DATA_BLOCK "METIS_AUX_DB"   // DB100
TITLE = Auxiliary help variables
{ S7_Optimized_Access := 'FALSE' }
AUTHOR : METIS
FAMILY : ACESYS
NAME : MiscDB
VERSION : 8.0
   VAR
      _REAL : Array[1..1000] of Real;   // Temporary REAL variables
      _INT : Array[1..200] of Int;   // Temporary INT variables
      _DINT : Array[1..200] of DInt;   // Temporary DINT variables
      _TIME : Array[1..100] of Time;   // Temporary TIME variables
      _BOOL : Array[1..512] of Bool;   // Temporary BOOLEAN variables
   END_VAR
BEGIN
   _REAL[1] := 8.0;
   _REAL[2] := 0.0;
   _REAL[3] := 16#FFC0_0000;
   _REAL[4] := 0.0;
   _REAL[5] := 0.0;
   _REAL[6] := 360.0;
   _REAL[7] := 1.0;
   _REAL[8] := 0.0;
   _REAL[9] := -32768.0;
   _REAL[10] := 0.0;
   _REAL[11] := 0.0;
   _REAL[12] := 0.0;
   _REAL[13] := 0.0;
   _REAL[14] := 0.0;
   _REAL[15] := 0.0;
   _REAL[16] := 0.0;
   _REAL[17] := 0.0;
   _REAL[18] := 0.0;
   _REAL[19] := 0.0;
   _REAL[20] := 0.0;
   _REAL[21] := 0.0;
   _REAL[22] := 0.0;
   _REAL[23] := 0.0;
   _REAL[24] := 0.0;
   _REAL[25] := 0.0;
   _REAL[26] := 0.0;
   _REAL[27] := 0.0;
   _REAL[28] := 0.0;
   _REAL[29] := 0.0;
   _REAL[30] := 0.0;
   _REAL[31] := 0.0;
   _REAL[32] := 0.0;
   _REAL[33] := 0.0;
   _REAL[34] := 0.0;
   _REAL[35] := 0.0;
   _REAL[36] := 0.0;
   _REAL[37] := 0.0;
   _REAL[38] := 0.0;
   _REAL[39] := 0.0;
   _REAL[40] := 0.0;
   _REAL[41] := 0.0;
   _REAL[42] := 0.0;
   _REAL[43] := 0.0;
   _REAL[44] := 0.0;
   _REAL[45] := 0.0;
   _REAL[46] := 0.0;
   _REAL[47] := 0.0;
   _REAL[48] := 0.0;
   _REAL[49] := 0.0;
   _REAL[50] := 0.0;
   _REAL[51] := 0.0;
   _REAL[52] := 0.0;
   _REAL[53] := 0.0;
   _REAL[54] := 0.0;
   _REAL[55] := 0.0;
   _REAL[56] := 0.0;
   _REAL[57] := 0.0;
   _REAL[58] := 0.0;
   _REAL[59] := 0.0;
   _REAL[60] := 0.0;
   _REAL[61] := 0.0;
   _REAL[62] := 0.0;
   _REAL[63] := 0.0;
   _REAL[64] := 0.0;
   _REAL[65] := 0.0;
   _REAL[66] := 0.0;
   _REAL[67] := 0.0;
   _REAL[68] := 0.0;
   _REAL[69] := 0.0;
   _REAL[70] := 0.0;
   _REAL[71] := 0.0;
   _REAL[72] := 0.0;
   _REAL[73] := 0.0;
   _REAL[74] := 0.0;
   _REAL[75] := 0.0;
   _REAL[76] := 0.0;
   _REAL[77] := 0.0;
   _REAL[78] := 0.0;
   _REAL[79] := 0.0;
   _REAL[80] := 0.0;
   _REAL[81] := 0.0;
   _REAL[82] := 0.0;
   _REAL[83] := 0.0;
   _REAL[84] := 0.0;
   _REAL[85] := 0.0;
   _REAL[86] := 0.0;
   _REAL[87] := 0.0;
   _REAL[88] := 0.0;
   _REAL[89] := 0.0;
   _REAL[90] := 0.0;
   _REAL[91] := 0.0;
   _REAL[92] := 0.0;
   _REAL[93] := 0.0;
   _REAL[94] := 0.0;
   _REAL[95] := 0.0;
   _REAL[96] := 0.0;
   _REAL[97] := 0.0;
   _REAL[98] := 0.0;
   _REAL[99] := 0.0;
   _REAL[100] := 0.0;
   _REAL[101] := 0.0;
   _REAL[102] := 0.0;
   _REAL[103] := 0.0;
   _REAL[104] := 0.0;
   _REAL[105] := 0.0;
   _REAL[106] := 0.0;
   _REAL[107] := 0.0;
   _REAL[108] := 0.0;
   _REAL[109] := 0.0;
   _REAL[110] := 0.0;
   _REAL[111] := 0.0;
   _REAL[112] := 0.0;
   _REAL[113] := 0.0;
   _REAL[114] := 0.0;
   _REAL[115] := 0.0;
   _REAL[116] := 0.0;
   _REAL[117] := 0.0;
   _REAL[118] := 0.0;
   _REAL[119] := 0.0;
   _REAL[120] := 0.0;
   _REAL[121] := 0.0;
   _REAL[122] := 0.0;
   _REAL[123] := 0.0;
   _REAL[124] := 0.0;
   _REAL[125] := 0.0;
   _REAL[126] := 0.0;
   _REAL[127] := 0.0;
   _REAL[128] := 0.0;
   _REAL[129] := 0.0;
   _REAL[130] := 0.0;
   _REAL[131] := 0.0;
   _REAL[132] := 0.0;
   _REAL[133] := 0.0;
   _REAL[134] := 0.0;
   _REAL[135] := 0.0;
   _REAL[136] := 0.0;
   _REAL[137] := 0.0;
   _REAL[138] := 0.0;
   _REAL[139] := 0.0;
   _REAL[140] := 0.0;
   _REAL[141] := 0.0;
   _REAL[142] := 0.0;
   _REAL[143] := 0.0;
   _REAL[144] := 0.0;
   _REAL[145] := 0.0;
   _REAL[146] := 0.0;
   _REAL[147] := 0.0;
   _REAL[148] := 0.0;
   _REAL[149] := 0.0;
   _REAL[150] := 0.0;
   _REAL[151] := 0.0;
   _REAL[152] := 0.0;
   _REAL[153] := 0.0;
   _REAL[154] := 0.0;
   _REAL[155] := 0.0;
   _REAL[156] := 0.0;
   _REAL[157] := 0.0;
   _REAL[158] := 0.0;
   _REAL[159] := 0.0;
   _REAL[160] := 0.0;
   _REAL[161] := 0.0;
   _REAL[162] := 0.0;
   _REAL[163] := 0.0;
   _REAL[164] := 0.0;
   _REAL[165] := 0.0;
   _REAL[166] := 0.0;
   _REAL[167] := 0.0;
   _REAL[168] := 0.0;
   _REAL[169] := 0.0;
   _REAL[170] := 0.0;
   _REAL[171] := 0.0;
   _REAL[172] := 0.0;
   _REAL[173] := 0.0;
   _REAL[174] := 0.0;
   _REAL[175] := 0.0;
   _REAL[176] := 0.0;
   _REAL[177] := 0.0;
   _REAL[178] := 0.0;
   _REAL[179] := 0.0;
   _REAL[180] := 0.0;
   _REAL[181] := 0.0;
   _REAL[182] := 0.0;
   _REAL[183] := 0.0;
   _REAL[184] := 0.0;
   _REAL[185] := 0.0;
   _REAL[186] := 0.0;
   _REAL[187] := 0.0;
   _REAL[188] := 0.0;
   _REAL[189] := 0.0;
   _REAL[190] := 0.0;
   _REAL[191] := 0.0;
   _REAL[192] := 0.0;
   _REAL[193] := 0.0;
   _REAL[194] := 0.0;
   _REAL[195] := 0.0;
   _REAL[196] := 0.0;
   _REAL[197] := 0.0;
   _REAL[198] := 0.0;
   _REAL[199] := 0.0;
   _REAL[200] := 0.0;
   _REAL[201] := 0.0;
   _REAL[202] := 0.0;
   _REAL[203] := 0.0;
   _REAL[204] := 0.0;
   _REAL[205] := 0.0;
   _REAL[206] := 0.0;
   _REAL[207] := 0.0;
   _REAL[208] := 0.0;
   _REAL[209] := 0.0;
   _REAL[210] := 0.0;
   _REAL[211] := 0.0;
   _REAL[212] := 0.0;
   _REAL[213] := 0.0;
   _REAL[214] := 0.0;
   _REAL[215] := 0.0;
   _REAL[216] := 0.0;
   _REAL[217] := 0.0;
   _REAL[218] := 0.0;
   _REAL[219] := 0.0;
   _REAL[220] := 0.0;
   _REAL[221] := 0.0;
   _REAL[222] := 0.0;
   _REAL[223] := 0.0;
   _REAL[224] := 0.0;
   _REAL[225] := 0.0;
   _REAL[226] := 0.0;
   _REAL[227] := 0.0;
   _REAL[228] := 0.0;
   _REAL[229] := 0.0;
   _REAL[230] := 0.0;
   _REAL[231] := 0.0;
   _REAL[232] := 0.0;
   _REAL[233] := 0.0;
   _REAL[234] := 0.0;
   _REAL[235] := 0.0;
   _REAL[236] := 0.0;
   _REAL[237] := 0.0;
   _REAL[238] := 0.0;
   _REAL[239] := 0.0;
   _REAL[240] := 0.0;
   _REAL[241] := 0.0;
   _REAL[242] := 0.0;
   _REAL[243] := 0.0;
   _REAL[244] := 0.0;
   _REAL[245] := 0.0;
   _REAL[246] := 0.0;
   _REAL[247] := 0.0;
   _REAL[248] := 0.0;
   _REAL[249] := 0.0;
   _REAL[250] := 0.0;
   _REAL[251] := 0.0;
   _REAL[252] := 0.0;
   _REAL[253] := 0.0;
   _REAL[254] := 0.0;
   _REAL[255] := 0.0;
   _REAL[256] := 0.0;
   _REAL[257] := 0.0;
   _REAL[258] := 0.0;
   _REAL[259] := 0.0;
   _REAL[260] := 0.0;
   _REAL[261] := 0.0;
   _REAL[262] := 0.0;
   _REAL[263] := 0.0;
   _REAL[264] := 0.0;
   _REAL[265] := 0.0;
   _REAL[266] := 0.0;
   _REAL[267] := 0.0;
   _REAL[268] := 0.0;
   _REAL[269] := 0.0;
   _REAL[270] := 0.0;
   _REAL[271] := 0.0;
   _REAL[272] := 0.0;
   _REAL[273] := 0.0;
   _REAL[274] := 0.0;
   _REAL[275] := 0.0;
   _REAL[276] := 0.0;
   _REAL[277] := 0.0;
   _REAL[278] := 0.0;
   _REAL[279] := 0.0;
   _REAL[280] := 0.0;
   _REAL[281] := 0.0;
   _REAL[282] := 0.0;
   _REAL[283] := 0.0;
   _REAL[284] := 0.0;
   _REAL[285] := 0.0;
   _REAL[286] := 0.0;
   _REAL[287] := 0.0;
   _REAL[288] := 0.0;
   _REAL[289] := 0.0;
   _REAL[290] := 0.0;
   _REAL[291] := 0.0;
   _REAL[292] := 0.0;
   _REAL[293] := 0.0;
   _REAL[294] := 0.0;
   _REAL[295] := 0.0;
   _REAL[296] := 0.0;
   _REAL[297] := 0.0;
   _REAL[298] := 0.0;
   _REAL[299] := 0.0;
   _REAL[300] := 0.0;
   _REAL[301] := 0.0;
   _REAL[302] := 0.0;
   _REAL[303] := 0.0;
   _REAL[304] := 0.0;
   _REAL[305] := 0.0;
   _REAL[306] := 0.0;
   _REAL[307] := 0.0;
   _REAL[308] := 0.0;
   _REAL[309] := 0.0;
   _REAL[310] := 0.0;
   _REAL[311] := 0.0;
   _REAL[312] := 0.0;
   _REAL[313] := 0.0;
   _REAL[314] := 0.0;
   _REAL[315] := 0.0;
   _REAL[316] := 0.0;
   _REAL[317] := 0.0;
   _REAL[318] := 0.0;
   _REAL[319] := 0.0;
   _REAL[320] := 0.0;
   _REAL[321] := 0.0;
   _REAL[322] := 0.0;
   _REAL[323] := 0.0;
   _REAL[324] := 0.0;
   _REAL[325] := 0.0;
   _REAL[326] := 0.0;
   _REAL[327] := 0.0;
   _REAL[328] := 0.0;
   _REAL[329] := 0.0;
   _REAL[330] := 0.0;
   _REAL[331] := 0.0;
   _REAL[332] := 0.0;
   _REAL[333] := 0.0;
   _REAL[334] := 0.0;
   _REAL[335] := 0.0;
   _REAL[336] := 0.0;
   _REAL[337] := 0.0;
   _REAL[338] := 0.0;
   _REAL[339] := 0.0;
   _REAL[340] := 0.0;
   _REAL[341] := 0.0;
   _REAL[342] := 0.0;
   _REAL[343] := 0.0;
   _REAL[344] := 0.0;
   _REAL[345] := 0.0;
   _REAL[346] := 0.0;
   _REAL[347] := 0.0;
   _REAL[348] := 0.0;
   _REAL[349] := 0.0;
   _REAL[350] := 0.0;
   _REAL[351] := 0.0;
   _REAL[352] := 0.0;
   _REAL[353] := 0.0;
   _REAL[354] := 0.0;
   _REAL[355] := 0.0;
   _REAL[356] := 0.0;
   _REAL[357] := 0.0;
   _REAL[358] := 0.0;
   _REAL[359] := 0.0;
   _REAL[360] := 0.0;
   _REAL[361] := 0.0;
   _REAL[362] := 0.0;
   _REAL[363] := 0.0;
   _REAL[364] := 0.0;
   _REAL[365] := 0.0;
   _REAL[366] := 0.0;
   _REAL[367] := 0.0;
   _REAL[368] := 0.0;
   _REAL[369] := 0.0;
   _REAL[370] := 0.0;
   _REAL[371] := 0.0;
   _REAL[372] := 0.0;
   _REAL[373] := 0.0;
   _REAL[374] := 0.0;
   _REAL[375] := 0.0;
   _REAL[376] := 0.0;
   _REAL[377] := 0.0;
   _REAL[378] := 0.0;
   _REAL[379] := 0.0;
   _REAL[380] := 0.0;
   _REAL[381] := 0.0;
   _REAL[382] := 0.0;
   _REAL[383] := 0.0;
   _REAL[384] := 0.0;
   _REAL[385] := 0.0;
   _REAL[386] := 0.0;
   _REAL[387] := 0.0;
   _REAL[388] := 0.0;
   _REAL[389] := 0.0;
   _REAL[390] := 0.0;
   _REAL[391] := 0.0;
   _REAL[392] := 0.0;
   _REAL[393] := 0.0;
   _REAL[394] := 0.0;
   _REAL[395] := 0.0;
   _REAL[396] := 0.0;
   _REAL[397] := 0.0;
   _REAL[398] := 0.0;
   _REAL[399] := 0.0;
   _REAL[400] := 0.0;
   _REAL[401] := 0.0;
   _REAL[402] := 0.0;
   _REAL[403] := 0.0;
   _REAL[404] := 0.0;
   _REAL[405] := 0.0;
   _REAL[406] := 0.0;
   _REAL[407] := 0.0;
   _REAL[408] := 0.0;
   _REAL[409] := 0.0;
   _REAL[410] := 0.0;
   _REAL[411] := 0.0;
   _REAL[412] := 0.0;
   _REAL[413] := 0.0;
   _REAL[414] := 0.0;
   _REAL[415] := 0.0;
   _REAL[416] := 0.0;
   _REAL[417] := 0.0;
   _REAL[418] := 0.0;
   _REAL[419] := 0.0;
   _REAL[420] := 0.0;
   _REAL[421] := 0.0;
   _REAL[422] := 0.0;
   _REAL[423] := 0.0;
   _REAL[424] := 0.0;
   _REAL[425] := 0.0;
   _REAL[426] := 0.0;
   _REAL[427] := 0.0;
   _REAL[428] := 0.0;
   _REAL[429] := 0.0;
   _REAL[430] := 0.0;
   _REAL[431] := 0.0;
   _REAL[432] := 0.0;
   _REAL[433] := 0.0;
   _REAL[434] := 0.0;
   _REAL[435] := 0.0;
   _REAL[436] := 0.0;
   _REAL[437] := 0.0;
   _REAL[438] := 0.0;
   _REAL[439] := 0.0;
   _REAL[440] := 0.0;
   _REAL[441] := 0.0;
   _REAL[442] := 0.0;
   _REAL[443] := 0.0;
   _REAL[444] := 0.0;
   _REAL[445] := 0.0;
   _REAL[446] := 0.0;
   _REAL[447] := 0.0;
   _REAL[448] := 0.0;
   _REAL[449] := 0.0;
   _REAL[450] := 0.0;
   _REAL[451] := 0.0;
   _REAL[452] := 0.0;
   _REAL[453] := 0.0;
   _REAL[454] := 0.0;
   _REAL[455] := 0.0;
   _REAL[456] := 0.0;
   _REAL[457] := 0.0;
   _REAL[458] := 0.0;
   _REAL[459] := 0.0;
   _REAL[460] := 0.0;
   _REAL[461] := 0.0;
   _REAL[462] := 0.0;
   _REAL[463] := 0.0;
   _REAL[464] := 0.0;
   _REAL[465] := 0.0;
   _REAL[466] := 0.0;
   _REAL[467] := 0.0;
   _REAL[468] := 0.0;
   _REAL[469] := 0.0;
   _REAL[470] := 0.0;
   _REAL[471] := 0.0;
   _REAL[472] := 0.0;
   _REAL[473] := 0.0;
   _REAL[474] := 0.0;
   _REAL[475] := 0.0;
   _REAL[476] := 0.0;
   _REAL[477] := 0.0;
   _REAL[478] := 0.0;
   _REAL[479] := 0.0;
   _REAL[480] := 0.0;
   _REAL[481] := 0.0;
   _REAL[482] := 0.0;
   _REAL[483] := 0.0;
   _REAL[484] := 0.0;
   _REAL[485] := 0.0;
   _REAL[486] := 0.0;
   _REAL[487] := 0.0;
   _REAL[488] := 0.0;
   _REAL[489] := 0.0;
   _REAL[490] := 0.0;
   _REAL[491] := 0.0;
   _REAL[492] := 0.0;
   _REAL[493] := 0.0;
   _REAL[494] := 0.0;
   _REAL[495] := 0.0;
   _REAL[496] := 0.0;
   _REAL[497] := 0.0;
   _REAL[498] := 0.0;
   _REAL[499] := 0.0;
   _REAL[500] := 0.0;
   _REAL[501] := 0.0;
   _REAL[502] := 0.0;
   _REAL[503] := 0.0;
   _REAL[504] := 0.0;
   _REAL[505] := 0.0;
   _REAL[506] := 0.0;
   _REAL[507] := 0.0;
   _REAL[508] := 0.0;
   _REAL[509] := 0.0;
   _REAL[510] := 0.0;
   _REAL[511] := 0.0;
   _REAL[512] := 0.0;
   _REAL[513] := 0.0;
   _REAL[514] := 0.0;
   _REAL[515] := 0.0;
   _REAL[516] := 0.0;
   _REAL[517] := 0.0;
   _REAL[518] := 0.0;
   _REAL[519] := 0.0;
   _REAL[520] := 0.0;
   _REAL[521] := 0.0;
   _REAL[522] := 0.0;
   _REAL[523] := 0.0;
   _REAL[524] := 0.0;
   _REAL[525] := 0.0;
   _REAL[526] := 0.0;
   _REAL[527] := 0.0;
   _REAL[528] := 0.0;
   _REAL[529] := 0.0;
   _REAL[530] := 0.0;
   _REAL[531] := 0.0;
   _REAL[532] := 0.0;
   _REAL[533] := 0.0;
   _REAL[534] := 0.0;
   _REAL[535] := 0.0;
   _REAL[536] := 0.0;
   _REAL[537] := 0.0;
   _REAL[538] := 0.0;
   _REAL[539] := 0.0;
   _REAL[540] := 0.0;
   _REAL[541] := 0.0;
   _REAL[542] := 0.0;
   _REAL[543] := 0.0;
   _REAL[544] := 0.0;
   _REAL[545] := 0.0;
   _REAL[546] := 0.0;
   _REAL[547] := 0.0;
   _REAL[548] := 0.0;
   _REAL[549] := 0.0;
   _REAL[550] := 0.0;
   _REAL[551] := 0.0;
   _REAL[552] := 0.0;
   _REAL[553] := 0.0;
   _REAL[554] := 0.0;
   _REAL[555] := 0.0;
   _REAL[556] := 0.0;
   _REAL[557] := 0.0;
   _REAL[558] := 0.0;
   _REAL[559] := 0.0;
   _REAL[560] := 0.0;
   _REAL[561] := 0.0;
   _REAL[562] := 0.0;
   _REAL[563] := 0.0;
   _REAL[564] := 0.0;
   _REAL[565] := 0.0;
   _REAL[566] := 0.0;
   _REAL[567] := 0.0;
   _REAL[568] := 0.0;
   _REAL[569] := 0.0;
   _REAL[570] := 0.0;
   _REAL[571] := 0.0;
   _REAL[572] := 0.0;
   _REAL[573] := 0.0;
   _REAL[574] := 0.0;
   _REAL[575] := 0.0;
   _REAL[576] := 0.0;
   _REAL[577] := 0.0;
   _REAL[578] := 0.0;
   _REAL[579] := 0.0;
   _REAL[580] := 0.0;
   _REAL[581] := 0.0;
   _REAL[582] := 0.0;
   _REAL[583] := 0.0;
   _REAL[584] := 0.0;
   _REAL[585] := 0.0;
   _REAL[586] := 0.0;
   _REAL[587] := 0.0;
   _REAL[588] := 0.0;
   _REAL[589] := 0.0;
   _REAL[590] := 0.0;
   _REAL[591] := 0.0;
   _REAL[592] := 0.0;
   _REAL[593] := 0.0;
   _REAL[594] := 0.0;
   _REAL[595] := 0.0;
   _REAL[596] := 0.0;
   _REAL[597] := 0.0;
   _REAL[598] := 0.0;
   _REAL[599] := 0.0;
   _REAL[600] := 0.0;
   _REAL[601] := 0.0;
   _REAL[602] := 0.0;
   _REAL[603] := 0.0;
   _REAL[604] := 0.0;
   _REAL[605] := 0.0;
   _REAL[606] := 0.0;
   _REAL[607] := 0.0;
   _REAL[608] := 0.0;
   _REAL[609] := 0.0;
   _REAL[610] := 0.0;
   _REAL[611] := 0.0;
   _REAL[612] := 0.0;
   _REAL[613] := 0.0;
   _REAL[614] := 0.0;
   _REAL[615] := 0.0;
   _REAL[616] := 0.0;
   _REAL[617] := 0.0;
   _REAL[618] := 0.0;
   _REAL[619] := 0.0;
   _REAL[620] := 0.0;
   _REAL[621] := 0.0;
   _REAL[622] := 0.0;
   _REAL[623] := 0.0;
   _REAL[624] := 0.0;
   _REAL[625] := 0.0;
   _REAL[626] := 0.0;
   _REAL[627] := 0.0;
   _REAL[628] := 0.0;
   _REAL[629] := 0.0;
   _REAL[630] := 0.0;
   _REAL[631] := 0.0;
   _REAL[632] := 0.0;
   _REAL[633] := 0.0;
   _REAL[634] := 0.0;
   _REAL[635] := 0.0;
   _REAL[636] := 0.0;
   _REAL[637] := 0.0;
   _REAL[638] := 0.0;
   _REAL[639] := 0.0;
   _REAL[640] := 0.0;
   _REAL[641] := 0.0;
   _REAL[642] := 0.0;
   _REAL[643] := 0.0;
   _REAL[644] := 0.0;
   _REAL[645] := 0.0;
   _REAL[646] := 0.0;
   _REAL[647] := 0.0;
   _REAL[648] := 0.0;
   _REAL[649] := 0.0;
   _REAL[650] := 0.0;
   _REAL[651] := 0.0;
   _REAL[652] := 0.0;
   _REAL[653] := 0.0;
   _REAL[654] := 0.0;
   _REAL[655] := 0.0;
   _REAL[656] := 0.0;
   _REAL[657] := 0.0;
   _REAL[658] := 0.0;
   _REAL[659] := 0.0;
   _REAL[660] := 0.0;
   _REAL[661] := 0.0;
   _REAL[662] := 0.0;
   _REAL[663] := 0.0;
   _REAL[664] := 0.0;
   _REAL[665] := 0.0;
   _REAL[666] := 0.0;
   _REAL[667] := 0.0;
   _REAL[668] := 0.0;
   _REAL[669] := 0.0;
   _REAL[670] := 0.0;
   _REAL[671] := 0.0;
   _REAL[672] := 0.0;
   _REAL[673] := 0.0;
   _REAL[674] := 0.0;
   _REAL[675] := 0.0;
   _REAL[676] := 0.0;
   _REAL[677] := 0.0;
   _REAL[678] := 0.0;
   _REAL[679] := 0.0;
   _REAL[680] := 0.0;
   _REAL[681] := 0.0;
   _REAL[682] := 0.0;
   _REAL[683] := 0.0;
   _REAL[684] := 0.0;
   _REAL[685] := 0.0;
   _REAL[686] := 0.0;
   _REAL[687] := 0.0;
   _REAL[688] := 0.0;
   _REAL[689] := 0.0;
   _REAL[690] := 0.0;
   _REAL[691] := 0.0;
   _REAL[692] := 0.0;
   _REAL[693] := 0.0;
   _REAL[694] := 0.0;
   _REAL[695] := 0.0;
   _REAL[696] := 0.0;
   _REAL[697] := 0.0;
   _REAL[698] := 0.0;
   _REAL[699] := 0.0;
   _REAL[700] := 0.0;
   _REAL[701] := 0.0;
   _REAL[702] := 0.0;
   _REAL[703] := 0.0;
   _REAL[704] := 0.0;
   _REAL[705] := 0.0;
   _REAL[706] := 0.0;
   _REAL[707] := 0.0;
   _REAL[708] := 0.0;
   _REAL[709] := 0.0;
   _REAL[710] := 0.0;
   _REAL[711] := 0.0;
   _REAL[712] := 0.0;
   _REAL[713] := 0.0;
   _REAL[714] := 0.0;
   _REAL[715] := 0.0;
   _REAL[716] := 0.0;
   _REAL[717] := 0.0;
   _REAL[718] := 0.0;
   _REAL[719] := 0.0;
   _REAL[720] := 0.0;
   _REAL[721] := 0.0;
   _REAL[722] := 0.0;
   _REAL[723] := 0.0;
   _REAL[724] := 0.0;
   _REAL[725] := 0.0;
   _REAL[726] := 0.0;
   _REAL[727] := 0.0;
   _REAL[728] := 0.0;
   _REAL[729] := 0.0;
   _REAL[730] := 0.0;
   _REAL[731] := 0.0;
   _REAL[732] := 0.0;
   _REAL[733] := 0.0;
   _REAL[734] := 0.0;
   _REAL[735] := 0.0;
   _REAL[736] := 0.0;
   _REAL[737] := 0.0;
   _REAL[738] := 0.0;
   _REAL[739] := 0.0;
   _REAL[740] := 0.0;
   _REAL[741] := 0.0;
   _REAL[742] := 0.0;
   _REAL[743] := 0.0;
   _REAL[744] := 0.0;
   _REAL[745] := 0.0;
   _REAL[746] := 0.0;
   _REAL[747] := 0.0;
   _REAL[748] := 0.0;
   _REAL[749] := 0.0;
   _REAL[750] := 0.0;
   _REAL[751] := 0.0;
   _REAL[752] := 0.0;
   _REAL[753] := 0.0;
   _REAL[754] := 0.0;
   _REAL[755] := 0.0;
   _REAL[756] := 0.0;
   _REAL[757] := 0.0;
   _REAL[758] := 0.0;
   _REAL[759] := 0.0;
   _REAL[760] := 0.0;
   _REAL[761] := 0.0;
   _REAL[762] := 0.0;
   _REAL[763] := 0.0;
   _REAL[764] := 0.0;
   _REAL[765] := 0.0;
   _REAL[766] := 0.0;
   _REAL[767] := 0.0;
   _REAL[768] := 0.0;
   _REAL[769] := 0.0;
   _REAL[770] := 0.0;
   _REAL[771] := 0.0;
   _REAL[772] := 0.0;
   _REAL[773] := 0.0;
   _REAL[774] := 0.0;
   _REAL[775] := 0.0;
   _REAL[776] := 0.0;
   _REAL[777] := 0.0;
   _REAL[778] := 0.0;
   _REAL[779] := 0.0;
   _REAL[780] := 0.0;
   _REAL[781] := 0.0;
   _REAL[782] := 0.0;
   _REAL[783] := 0.0;
   _REAL[784] := 0.0;
   _REAL[785] := 0.0;
   _REAL[786] := 0.0;
   _REAL[787] := 0.0;
   _REAL[788] := 0.0;
   _REAL[789] := 0.0;
   _REAL[790] := 0.0;
   _REAL[791] := 0.0;
   _REAL[792] := 0.0;
   _REAL[793] := 0.0;
   _REAL[794] := 0.0;
   _REAL[795] := 0.0;
   _REAL[796] := 0.0;
   _REAL[797] := 0.0;
   _REAL[798] := 0.0;
   _REAL[799] := 0.0;
   _REAL[800] := 0.0;
   _REAL[801] := 0.0;
   _REAL[802] := 0.0;
   _REAL[803] := 0.0;
   _REAL[804] := 0.0;
   _REAL[805] := 0.0;
   _REAL[806] := 0.0;
   _REAL[807] := 0.0;
   _REAL[808] := 0.0;
   _REAL[809] := 0.0;
   _REAL[810] := 0.0;
   _REAL[811] := 0.0;
   _REAL[812] := 0.0;
   _REAL[813] := 0.0;
   _REAL[814] := 0.0;
   _REAL[815] := 0.0;
   _REAL[816] := 0.0;
   _REAL[817] := 0.0;
   _REAL[818] := 0.0;
   _REAL[819] := 0.0;
   _REAL[820] := 0.0;
   _REAL[821] := 0.0;
   _REAL[822] := 0.0;
   _REAL[823] := 0.0;
   _REAL[824] := 0.0;
   _REAL[825] := 0.0;
   _REAL[826] := 0.0;
   _REAL[827] := 0.0;
   _REAL[828] := 0.0;
   _REAL[829] := 0.0;
   _REAL[830] := 0.0;
   _REAL[831] := 0.0;
   _REAL[832] := 0.0;
   _REAL[833] := 0.0;
   _REAL[834] := 0.0;
   _REAL[835] := 0.0;
   _REAL[836] := 0.0;
   _REAL[837] := 0.0;
   _REAL[838] := 0.0;
   _REAL[839] := 0.0;
   _REAL[840] := 0.0;
   _REAL[841] := 0.0;
   _REAL[842] := 0.0;
   _REAL[843] := 0.0;
   _REAL[844] := 0.0;
   _REAL[845] := 0.0;
   _REAL[846] := 0.0;
   _REAL[847] := 0.0;
   _REAL[848] := 0.0;
   _REAL[849] := 0.0;
   _REAL[850] := 0.0;
   _REAL[851] := 0.0;
   _REAL[852] := 0.0;
   _REAL[853] := 0.0;
   _REAL[854] := 0.0;
   _REAL[855] := 0.0;
   _REAL[856] := 0.0;
   _REAL[857] := 0.0;
   _REAL[858] := 0.0;
   _REAL[859] := 0.0;
   _REAL[860] := 0.0;
   _REAL[861] := 0.0;
   _REAL[862] := 0.0;
   _REAL[863] := 0.0;
   _REAL[864] := 0.0;
   _REAL[865] := 0.0;
   _REAL[866] := 0.0;
   _REAL[867] := 0.0;
   _REAL[868] := 0.0;
   _REAL[869] := 0.0;
   _REAL[870] := 0.0;
   _REAL[871] := 0.0;
   _REAL[872] := 0.0;
   _REAL[873] := 0.0;
   _REAL[874] := 0.0;
   _REAL[875] := 0.0;
   _REAL[876] := 0.0;
   _REAL[877] := 0.0;
   _REAL[878] := 0.0;
   _REAL[879] := 0.0;
   _REAL[880] := 0.0;
   _REAL[881] := 0.0;
   _REAL[882] := 0.0;
   _REAL[883] := 0.0;
   _REAL[884] := 0.0;
   _REAL[885] := 0.0;
   _REAL[886] := 0.0;
   _REAL[887] := 0.0;
   _REAL[888] := 0.0;
   _REAL[889] := 0.0;
   _REAL[890] := 0.0;
   _REAL[891] := 0.0;
   _REAL[892] := 0.0;
   _REAL[893] := 0.0;
   _REAL[894] := 0.0;
   _REAL[895] := 0.0;
   _REAL[896] := 0.0;
   _REAL[897] := 0.0;
   _REAL[898] := 0.0;
   _REAL[899] := 0.0;
   _REAL[900] := 0.0;
   _REAL[901] := 0.0;
   _REAL[902] := 0.0;
   _REAL[903] := 0.0;
   _REAL[904] := 0.0;
   _REAL[905] := 0.0;
   _REAL[906] := 0.0;
   _REAL[907] := 0.0;
   _REAL[908] := 0.0;
   _REAL[909] := 0.0;
   _REAL[910] := 0.0;
   _REAL[911] := 0.0;
   _REAL[912] := 0.0;
   _REAL[913] := 0.0;
   _REAL[914] := 0.0;
   _REAL[915] := 0.0;
   _REAL[916] := 0.0;
   _REAL[917] := 0.0;
   _REAL[918] := 0.0;
   _REAL[919] := 0.0;
   _REAL[920] := 0.0;
   _REAL[921] := 0.0;
   _REAL[922] := 0.0;
   _REAL[923] := 0.0;
   _REAL[924] := 0.0;
   _REAL[925] := 0.0;
   _REAL[926] := 0.0;
   _REAL[927] := 0.0;
   _REAL[928] := 0.0;
   _REAL[929] := 0.0;
   _REAL[930] := 0.0;
   _REAL[931] := 0.0;
   _REAL[932] := 0.0;
   _REAL[933] := 0.0;
   _REAL[934] := 0.0;
   _REAL[935] := 0.0;
   _REAL[936] := 0.0;
   _REAL[937] := 0.0;
   _REAL[938] := 0.0;
   _REAL[939] := 0.0;
   _REAL[940] := 0.0;
   _REAL[941] := 0.0;
   _REAL[942] := 0.0;
   _REAL[943] := 0.0;
   _REAL[944] := 0.0;
   _REAL[945] := 0.0;
   _REAL[946] := 0.0;
   _REAL[947] := 0.0;
   _REAL[948] := 0.0;
   _REAL[949] := 0.0;
   _REAL[950] := 0.0;
   _REAL[951] := 0.0;
   _REAL[952] := 0.0;
   _REAL[953] := 0.0;
   _REAL[954] := 0.0;
   _REAL[955] := 0.0;
   _REAL[956] := 0.0;
   _REAL[957] := 0.0;
   _REAL[958] := 0.0;
   _REAL[959] := 0.0;
   _REAL[960] := 0.0;
   _REAL[961] := 0.0;
   _REAL[962] := 0.0;
   _REAL[963] := 0.0;
   _REAL[964] := 0.0;
   _REAL[965] := 0.0;
   _REAL[966] := 0.0;
   _REAL[967] := 0.0;
   _REAL[968] := 0.0;
   _REAL[969] := 0.0;
   _REAL[970] := 0.0;
   _REAL[971] := 0.0;
   _REAL[972] := 0.0;
   _REAL[973] := 0.0;
   _REAL[974] := 0.0;
   _REAL[975] := 0.0;
   _REAL[976] := 0.0;
   _REAL[977] := 0.0;
   _REAL[978] := 0.0;
   _REAL[979] := 0.0;
   _REAL[980] := 0.0;
   _REAL[981] := 0.0;
   _REAL[982] := 0.0;
   _REAL[983] := 0.0;
   _REAL[984] := 0.0;
   _REAL[985] := 0.0;
   _REAL[986] := 0.0;
   _REAL[987] := 0.0;
   _REAL[988] := 0.0;
   _REAL[989] := 0.0;
   _REAL[990] := 0.0;
   _REAL[991] := 0.0;
   _REAL[992] := 0.0;
   _REAL[993] := 0.0;
   _REAL[994] := 0.0;
   _REAL[995] := 0.0;
   _REAL[996] := 0.0;
   _REAL[997] := 0.0;
   _REAL[998] := 0.0;
   _REAL[999] := 0.0;
   _REAL[1000] := 0.0;
   _INT[1] := 0;
   _INT[2] := 0;
   _INT[3] := 0;
   _INT[4] := 0;
   _INT[5] := 0;
   _INT[6] := 0;
   _INT[7] := 0;
   _INT[8] := 0;
   _INT[9] := 0;
   _INT[10] := 0;
   _INT[11] := 0;
   _INT[12] := 0;
   _INT[13] := 0;
   _INT[14] := 0;
   _INT[15] := 0;
   _INT[16] := 0;
   _INT[17] := 0;
   _INT[18] := 0;
   _INT[19] := 0;
   _INT[20] := 0;
   _INT[21] := 0;
   _INT[22] := 0;
   _INT[23] := 0;
   _INT[24] := 0;
   _INT[25] := 0;
   _INT[26] := 0;
   _INT[27] := 0;
   _INT[28] := 0;
   _INT[29] := 0;
   _INT[30] := 0;
   _INT[31] := 0;
   _INT[32] := 0;
   _INT[33] := 0;
   _INT[34] := 0;
   _INT[35] := 0;
   _INT[36] := 0;
   _INT[37] := 0;
   _INT[38] := 0;
   _INT[39] := 0;
   _INT[40] := 0;
   _INT[41] := 0;
   _INT[42] := 0;
   _INT[43] := 0;
   _INT[44] := 0;
   _INT[45] := 0;
   _INT[46] := 0;
   _INT[47] := 0;
   _INT[48] := 0;
   _INT[49] := 0;
   _INT[50] := 0;
   _INT[51] := 0;
   _INT[52] := 0;
   _INT[53] := 0;
   _INT[54] := 0;
   _INT[55] := 0;
   _INT[56] := 0;
   _INT[57] := 0;
   _INT[58] := 0;
   _INT[59] := 0;
   _INT[60] := 0;
   _INT[61] := 0;
   _INT[62] := 0;
   _INT[63] := 0;
   _INT[64] := 0;
   _INT[65] := 0;
   _INT[66] := 0;
   _INT[67] := 0;
   _INT[68] := 0;
   _INT[69] := 0;
   _INT[70] := 0;
   _INT[71] := 0;
   _INT[72] := 0;
   _INT[73] := 0;
   _INT[74] := 0;
   _INT[75] := 0;
   _INT[76] := 0;
   _INT[77] := 0;
   _INT[78] := 0;
   _INT[79] := 0;
   _INT[80] := 0;
   _INT[81] := 0;
   _INT[82] := 0;
   _INT[83] := 0;
   _INT[84] := 0;
   _INT[85] := 0;
   _INT[86] := 0;
   _INT[87] := 0;
   _INT[88] := 0;
   _INT[89] := 0;
   _INT[90] := 0;
   _INT[91] := 0;
   _INT[92] := 0;
   _INT[93] := 0;
   _INT[94] := 0;
   _INT[95] := 0;
   _INT[96] := 0;
   _INT[97] := 0;
   _INT[98] := 0;
   _INT[99] := 0;
   _INT[100] := 0;
   _INT[101] := 0;
   _INT[102] := 0;
   _INT[103] := 0;
   _INT[104] := 0;
   _INT[105] := 0;
   _INT[106] := 0;
   _INT[107] := 0;
   _INT[108] := 0;
   _INT[109] := 0;
   _INT[110] := 0;
   _INT[111] := 0;
   _INT[112] := 0;
   _INT[113] := 0;
   _INT[114] := 0;
   _INT[115] := 0;
   _INT[116] := 0;
   _INT[117] := 0;
   _INT[118] := 0;
   _INT[119] := 0;
   _INT[120] := 0;
   _INT[121] := 0;
   _INT[122] := 0;
   _INT[123] := 0;
   _INT[124] := 0;
   _INT[125] := 0;
   _INT[126] := 0;
   _INT[127] := 0;
   _INT[128] := 0;
   _INT[129] := 0;
   _INT[130] := 0;
   _INT[131] := 0;
   _INT[132] := 0;
   _INT[133] := 0;
   _INT[134] := 0;
   _INT[135] := 0;
   _INT[136] := 0;
   _INT[137] := 0;
   _INT[138] := 0;
   _INT[139] := 0;
   _INT[140] := 0;
   _INT[141] := 0;
   _INT[142] := 0;
   _INT[143] := 0;
   _INT[144] := 0;
   _INT[145] := 0;
   _INT[146] := 0;
   _INT[147] := 0;
   _INT[148] := 0;
   _INT[149] := 0;
   _INT[150] := 0;
   _INT[151] := 0;
   _INT[152] := 0;
   _INT[153] := 0;
   _INT[154] := 0;
   _INT[155] := 0;
   _INT[156] := 0;
   _INT[157] := 0;
   _INT[158] := 0;
   _INT[159] := 0;
   _INT[160] := 0;
   _INT[161] := 0;
   _INT[162] := 0;
   _INT[163] := 0;
   _INT[164] := 0;
   _INT[165] := 0;
   _INT[166] := 0;
   _INT[167] := 0;
   _INT[168] := 0;
   _INT[169] := 0;
   _INT[170] := 0;
   _INT[171] := 0;
   _INT[172] := 0;
   _INT[173] := 0;
   _INT[174] := 0;
   _INT[175] := 0;
   _INT[176] := 0;
   _INT[177] := 0;
   _INT[178] := 0;
   _INT[179] := 0;
   _INT[180] := 0;
   _INT[181] := 0;
   _INT[182] := 0;
   _INT[183] := 0;
   _INT[184] := 0;
   _INT[185] := 0;
   _INT[186] := 0;
   _INT[187] := 0;
   _INT[188] := 0;
   _INT[189] := 0;
   _INT[190] := 0;
   _INT[191] := 0;
   _INT[192] := 0;
   _INT[193] := 0;
   _INT[194] := 0;
   _INT[195] := 0;
   _INT[196] := 0;
   _INT[197] := 0;
   _INT[198] := 0;
   _INT[199] := 0;
   _INT[200] := 0;
   _DINT[1] := 0;
   _DINT[2] := 0;
   _DINT[3] := 0;
   _DINT[4] := 0;
   _DINT[5] := 0;
   _DINT[6] := 0;
   _DINT[7] := 0;
   _DINT[8] := 0;
   _DINT[9] := 0;
   _DINT[10] := 0;
   _DINT[11] := 0;
   _DINT[12] := 0;
   _DINT[13] := 0;
   _DINT[14] := 0;
   _DINT[15] := 0;
   _DINT[16] := 0;
   _DINT[17] := 0;
   _DINT[18] := 0;
   _DINT[19] := 0;
   _DINT[20] := 0;
   _DINT[21] := 0;
   _DINT[22] := 0;
   _DINT[23] := 0;
   _DINT[24] := 0;
   _DINT[25] := 0;
   _DINT[26] := 0;
   _DINT[27] := 0;
   _DINT[28] := 0;
   _DINT[29] := 0;
   _DINT[30] := 0;
   _DINT[31] := 0;
   _DINT[32] := 0;
   _DINT[33] := 0;
   _DINT[34] := 0;
   _DINT[35] := 0;
   _DINT[36] := 0;
   _DINT[37] := 0;
   _DINT[38] := 0;
   _DINT[39] := 0;
   _DINT[40] := 0;
   _DINT[41] := 0;
   _DINT[42] := 0;
   _DINT[43] := 0;
   _DINT[44] := 0;
   _DINT[45] := 0;
   _DINT[46] := 0;
   _DINT[47] := 0;
   _DINT[48] := 0;
   _DINT[49] := 0;
   _DINT[50] := 0;
   _DINT[51] := 0;
   _DINT[52] := 0;
   _DINT[53] := 0;
   _DINT[54] := 0;
   _DINT[55] := 0;
   _DINT[56] := 0;
   _DINT[57] := 0;
   _DINT[58] := 0;
   _DINT[59] := 0;
   _DINT[60] := 0;
   _DINT[61] := 0;
   _DINT[62] := 0;
   _DINT[63] := 0;
   _DINT[64] := 0;
   _DINT[65] := 0;
   _DINT[66] := 0;
   _DINT[67] := 0;
   _DINT[68] := 0;
   _DINT[69] := 0;
   _DINT[70] := 0;
   _DINT[71] := 0;
   _DINT[72] := 0;
   _DINT[73] := 0;
   _DINT[74] := 0;
   _DINT[75] := 0;
   _DINT[76] := 0;
   _DINT[77] := 0;
   _DINT[78] := 0;
   _DINT[79] := 0;
   _DINT[80] := 0;
   _DINT[81] := 0;
   _DINT[82] := 0;
   _DINT[83] := 0;
   _DINT[84] := 0;
   _DINT[85] := 0;
   _DINT[86] := 0;
   _DINT[87] := 0;
   _DINT[88] := 0;
   _DINT[89] := 0;
   _DINT[90] := 0;
   _DINT[91] := 0;
   _DINT[92] := 0;
   _DINT[93] := 0;
   _DINT[94] := 0;
   _DINT[95] := 0;
   _DINT[96] := 0;
   _DINT[97] := 0;
   _DINT[98] := 0;
   _DINT[99] := 0;
   _DINT[100] := 0;
   _DINT[101] := 0;
   _DINT[102] := 0;
   _DINT[103] := 0;
   _DINT[104] := 0;
   _DINT[105] := 0;
   _DINT[106] := 0;
   _DINT[107] := 0;
   _DINT[108] := 0;
   _DINT[109] := 0;
   _DINT[110] := 0;
   _DINT[111] := 0;
   _DINT[112] := 0;
   _DINT[113] := 0;
   _DINT[114] := 0;
   _DINT[115] := 0;
   _DINT[116] := 0;
   _DINT[117] := 0;
   _DINT[118] := 0;
   _DINT[119] := 0;
   _DINT[120] := 0;
   _DINT[121] := 0;
   _DINT[122] := 0;
   _DINT[123] := 0;
   _DINT[124] := 0;
   _DINT[125] := 0;
   _DINT[126] := 0;
   _DINT[127] := 0;
   _DINT[128] := 0;
   _DINT[129] := 0;
   _DINT[130] := 0;
   _DINT[131] := 0;
   _DINT[132] := 0;
   _DINT[133] := 0;
   _DINT[134] := 0;
   _DINT[135] := 0;
   _DINT[136] := 0;
   _DINT[137] := 0;
   _DINT[138] := 0;
   _DINT[139] := 0;
   _DINT[140] := 0;
   _DINT[141] := 0;
   _DINT[142] := 0;
   _DINT[143] := 0;
   _DINT[144] := 0;
   _DINT[145] := 0;
   _DINT[146] := 0;
   _DINT[147] := 0;
   _DINT[148] := 0;
   _DINT[149] := 0;
   _DINT[150] := 0;
   _DINT[151] := 0;
   _DINT[152] := 0;
   _DINT[153] := 0;
   _DINT[154] := 0;
   _DINT[155] := 0;
   _DINT[156] := 0;
   _DINT[157] := 0;
   _DINT[158] := 0;
   _DINT[159] := 0;
   _DINT[160] := 0;
   _DINT[161] := 0;
   _DINT[162] := 0;
   _DINT[163] := 0;
   _DINT[164] := 0;
   _DINT[165] := 0;
   _DINT[166] := 0;
   _DINT[167] := 0;
   _DINT[168] := 0;
   _DINT[169] := 0;
   _DINT[170] := 0;
   _DINT[171] := 0;
   _DINT[172] := 0;
   _DINT[173] := 0;
   _DINT[174] := 0;
   _DINT[175] := 0;
   _DINT[176] := 0;
   _DINT[177] := 0;
   _DINT[178] := 0;
   _DINT[179] := 0;
   _DINT[180] := 0;
   _DINT[181] := 0;
   _DINT[182] := 0;
   _DINT[183] := 0;
   _DINT[184] := 0;
   _DINT[185] := 0;
   _DINT[186] := 0;
   _DINT[187] := 0;
   _DINT[188] := 0;
   _DINT[189] := 0;
   _DINT[190] := 0;
   _DINT[191] := 0;
   _DINT[192] := 0;
   _DINT[193] := 0;
   _DINT[194] := 0;
   _DINT[195] := 0;
   _DINT[196] := 0;
   _DINT[197] := 0;
   _DINT[198] := 0;
   _DINT[199] := 0;
   _DINT[200] := 0;
   _TIME[1] := T#0MS;
   _TIME[2] := T#0MS;
   _TIME[3] := T#0MS;
   _TIME[4] := T#0MS;
   _TIME[5] := T#0MS;
   _TIME[6] := T#0MS;
   _TIME[7] := T#0MS;
   _TIME[8] := T#0MS;
   _TIME[9] := T#0MS;
   _TIME[10] := T#0MS;
   _TIME[11] := T#0MS;
   _TIME[12] := T#0MS;
   _TIME[13] := T#0MS;
   _TIME[14] := T#0MS;
   _TIME[15] := T#0MS;
   _TIME[16] := T#0MS;
   _TIME[17] := T#0MS;
   _TIME[18] := T#0MS;
   _TIME[19] := T#0MS;
   _TIME[20] := T#0MS;
   _TIME[21] := T#0MS;
   _TIME[22] := T#0MS;
   _TIME[23] := T#0MS;
   _TIME[24] := T#0MS;
   _TIME[25] := T#0MS;
   _TIME[26] := T#0MS;
   _TIME[27] := T#0MS;
   _TIME[28] := T#0MS;
   _TIME[29] := T#0MS;
   _TIME[30] := T#0MS;
   _TIME[31] := T#0MS;
   _TIME[32] := T#0MS;
   _TIME[33] := T#0MS;
   _TIME[34] := T#0MS;
   _TIME[35] := T#0MS;
   _TIME[36] := T#0MS;
   _TIME[37] := T#0MS;
   _TIME[38] := T#0MS;
   _TIME[39] := T#0MS;
   _TIME[40] := T#0MS;
   _TIME[41] := T#0MS;
   _TIME[42] := T#0MS;
   _TIME[43] := T#0MS;
   _TIME[44] := T#0MS;
   _TIME[45] := T#0MS;
   _TIME[46] := T#0MS;
   _TIME[47] := T#0MS;
   _TIME[48] := T#0MS;
   _TIME[49] := T#0MS;
   _TIME[50] := T#0MS;
   _TIME[51] := T#0MS;
   _TIME[52] := T#0MS;
   _TIME[53] := T#0MS;
   _TIME[54] := T#0MS;
   _TIME[55] := T#0MS;
   _TIME[56] := T#0MS;
   _TIME[57] := T#0MS;
   _TIME[58] := T#0MS;
   _TIME[59] := T#0MS;
   _TIME[60] := T#0MS;
   _TIME[61] := T#0MS;
   _TIME[62] := T#0MS;
   _TIME[63] := T#0MS;
   _TIME[64] := T#0MS;
   _TIME[65] := T#0MS;
   _TIME[66] := T#0MS;
   _TIME[67] := T#0MS;
   _TIME[68] := T#0MS;
   _TIME[69] := T#0MS;
   _TIME[70] := T#0MS;
   _TIME[71] := T#0MS;
   _TIME[72] := T#0MS;
   _TIME[73] := T#0MS;
   _TIME[74] := T#0MS;
   _TIME[75] := T#0MS;
   _TIME[76] := T#0MS;
   _TIME[77] := T#0MS;
   _TIME[78] := T#0MS;
   _TIME[79] := T#0MS;
   _TIME[80] := T#0MS;
   _TIME[81] := T#0MS;
   _TIME[82] := T#0MS;
   _TIME[83] := T#0MS;
   _TIME[84] := T#0MS;
   _TIME[85] := T#0MS;
   _TIME[86] := T#0MS;
   _TIME[87] := T#0MS;
   _TIME[88] := T#0MS;
   _TIME[89] := T#0MS;
   _TIME[90] := T#0MS;
   _TIME[91] := T#0MS;
   _TIME[92] := T#0MS;
   _TIME[93] := T#0MS;
   _TIME[94] := T#0MS;
   _TIME[95] := T#0MS;
   _TIME[96] := T#0MS;
   _TIME[97] := T#0MS;
   _TIME[98] := T#0MS;
   _TIME[99] := T#0MS;
   _TIME[100] := T#0MS;
   _BOOL[1] := FALSE;
   _BOOL[2] := FALSE;
   _BOOL[3] := FALSE;
   _BOOL[4] := FALSE;
   _BOOL[5] := FALSE;
   _BOOL[6] := FALSE;
   _BOOL[7] := FALSE;
   _BOOL[8] := FALSE;
   _BOOL[9] := FALSE;
   _BOOL[10] := FALSE;
   _BOOL[11] := FALSE;
   _BOOL[12] := FALSE;
   _BOOL[13] := FALSE;
   _BOOL[14] := FALSE;
   _BOOL[15] := FALSE;
   _BOOL[16] := FALSE;
   _BOOL[17] := FALSE;
   _BOOL[18] := FALSE;
   _BOOL[19] := FALSE;
   _BOOL[20] := FALSE;
   _BOOL[21] := FALSE;
   _BOOL[22] := FALSE;
   _BOOL[23] := FALSE;
   _BOOL[24] := FALSE;
   _BOOL[25] := FALSE;
   _BOOL[26] := FALSE;
   _BOOL[27] := FALSE;
   _BOOL[28] := FALSE;
   _BOOL[29] := FALSE;
   _BOOL[30] := FALSE;
   _BOOL[31] := FALSE;
   _BOOL[32] := FALSE;
   _BOOL[33] := FALSE;
   _BOOL[34] := FALSE;
   _BOOL[35] := FALSE;
   _BOOL[36] := FALSE;
   _BOOL[37] := FALSE;
   _BOOL[38] := FALSE;
   _BOOL[39] := FALSE;
   _BOOL[40] := FALSE;
   _BOOL[41] := FALSE;
   _BOOL[42] := FALSE;
   _BOOL[43] := FALSE;
   _BOOL[44] := FALSE;
   _BOOL[45] := FALSE;
   _BOOL[46] := FALSE;
   _BOOL[47] := FALSE;
   _BOOL[48] := FALSE;
   _BOOL[49] := FALSE;
   _BOOL[50] := FALSE;
   _BOOL[51] := FALSE;
   _BOOL[52] := FALSE;
   _BOOL[53] := FALSE;
   _BOOL[54] := FALSE;
   _BOOL[55] := FALSE;
   _BOOL[56] := FALSE;
   _BOOL[57] := FALSE;
   _BOOL[58] := FALSE;
   _BOOL[59] := FALSE;
   _BOOL[60] := FALSE;
   _BOOL[61] := FALSE;
   _BOOL[62] := FALSE;
   _BOOL[63] := FALSE;
   _BOOL[64] := FALSE;
   _BOOL[65] := FALSE;
   _BOOL[66] := FALSE;
   _BOOL[67] := FALSE;
   _BOOL[68] := FALSE;
   _BOOL[69] := FALSE;
   _BOOL[70] := FALSE;
   _BOOL[71] := FALSE;
   _BOOL[72] := FALSE;
   _BOOL[73] := FALSE;
   _BOOL[74] := FALSE;
   _BOOL[75] := FALSE;
   _BOOL[76] := FALSE;
   _BOOL[77] := FALSE;
   _BOOL[78] := FALSE;
   _BOOL[79] := FALSE;
   _BOOL[80] := FALSE;
   _BOOL[81] := FALSE;
   _BOOL[82] := FALSE;
   _BOOL[83] := FALSE;
   _BOOL[84] := FALSE;
   _BOOL[85] := FALSE;
   _BOOL[86] := FALSE;
   _BOOL[87] := FALSE;
   _BOOL[88] := FALSE;
   _BOOL[89] := FALSE;
   _BOOL[90] := FALSE;
   _BOOL[91] := FALSE;
   _BOOL[92] := FALSE;
   _BOOL[93] := FALSE;
   _BOOL[94] := FALSE;
   _BOOL[95] := FALSE;
   _BOOL[96] := FALSE;
   _BOOL[97] := FALSE;
   _BOOL[98] := FALSE;
   _BOOL[99] := FALSE;
   _BOOL[100] := FALSE;
   _BOOL[101] := FALSE;
   _BOOL[102] := FALSE;
   _BOOL[103] := FALSE;
   _BOOL[104] := FALSE;
   _BOOL[105] := FALSE;
   _BOOL[106] := FALSE;
   _BOOL[107] := FALSE;
   _BOOL[108] := FALSE;
   _BOOL[109] := FALSE;
   _BOOL[110] := FALSE;
   _BOOL[111] := FALSE;
   _BOOL[112] := FALSE;
   _BOOL[113] := FALSE;
   _BOOL[114] := FALSE;
   _BOOL[115] := FALSE;
   _BOOL[116] := FALSE;
   _BOOL[117] := FALSE;
   _BOOL[118] := FALSE;
   _BOOL[119] := FALSE;
   _BOOL[120] := FALSE;
   _BOOL[121] := FALSE;
   _BOOL[122] := FALSE;
   _BOOL[123] := FALSE;
   _BOOL[124] := FALSE;
   _BOOL[125] := FALSE;
   _BOOL[126] := FALSE;
   _BOOL[127] := FALSE;
   _BOOL[128] := FALSE;
   _BOOL[129] := FALSE;
   _BOOL[130] := FALSE;
   _BOOL[131] := FALSE;
   _BOOL[132] := FALSE;
   _BOOL[133] := FALSE;
   _BOOL[134] := FALSE;
   _BOOL[135] := FALSE;
   _BOOL[136] := FALSE;
   _BOOL[137] := FALSE;
   _BOOL[138] := FALSE;
   _BOOL[139] := FALSE;
   _BOOL[140] := FALSE;
   _BOOL[141] := FALSE;
   _BOOL[142] := FALSE;
   _BOOL[143] := FALSE;
   _BOOL[144] := FALSE;
   _BOOL[145] := FALSE;
   _BOOL[146] := FALSE;
   _BOOL[147] := FALSE;
   _BOOL[148] := FALSE;
   _BOOL[149] := FALSE;
   _BOOL[150] := FALSE;
   _BOOL[151] := FALSE;
   _BOOL[152] := FALSE;
   _BOOL[153] := FALSE;
   _BOOL[154] := FALSE;
   _BOOL[155] := FALSE;
   _BOOL[156] := FALSE;
   _BOOL[157] := FALSE;
   _BOOL[158] := FALSE;
   _BOOL[159] := FALSE;
   _BOOL[160] := FALSE;
   _BOOL[161] := FALSE;
   _BOOL[162] := FALSE;
   _BOOL[163] := FALSE;
   _BOOL[164] := FALSE;
   _BOOL[165] := FALSE;
   _BOOL[166] := FALSE;
   _BOOL[167] := FALSE;
   _BOOL[168] := FALSE;
   _BOOL[169] := FALSE;
   _BOOL[170] := FALSE;
   _BOOL[171] := FALSE;
   _BOOL[172] := FALSE;
   _BOOL[173] := FALSE;
   _BOOL[174] := FALSE;
   _BOOL[175] := FALSE;
   _BOOL[176] := FALSE;
   _BOOL[177] := FALSE;
   _BOOL[178] := FALSE;
   _BOOL[179] := FALSE;
   _BOOL[180] := FALSE;
   _BOOL[181] := FALSE;
   _BOOL[182] := FALSE;
   _BOOL[183] := FALSE;
   _BOOL[184] := FALSE;
   _BOOL[185] := FALSE;
   _BOOL[186] := FALSE;
   _BOOL[187] := FALSE;
   _BOOL[188] := FALSE;
   _BOOL[189] := FALSE;
   _BOOL[190] := FALSE;
   _BOOL[191] := FALSE;
   _BOOL[192] := FALSE;
   _BOOL[193] := FALSE;
   _BOOL[194] := FALSE;
   _BOOL[195] := FALSE;
   _BOOL[196] := FALSE;
   _BOOL[197] := FALSE;
   _BOOL[198] := FALSE;
   _BOOL[199] := FALSE;
   _BOOL[200] := FALSE;
   _BOOL[201] := FALSE;
   _BOOL[202] := FALSE;
   _BOOL[203] := FALSE;
   _BOOL[204] := FALSE;
   _BOOL[205] := FALSE;
   _BOOL[206] := FALSE;
   _BOOL[207] := FALSE;
   _BOOL[208] := FALSE;
   _BOOL[209] := FALSE;
   _BOOL[210] := FALSE;
   _BOOL[211] := FALSE;
   _BOOL[212] := FALSE;
   _BOOL[213] := FALSE;
   _BOOL[214] := FALSE;
   _BOOL[215] := FALSE;
   _BOOL[216] := FALSE;
   _BOOL[217] := FALSE;
   _BOOL[218] := FALSE;
   _BOOL[219] := FALSE;
   _BOOL[220] := FALSE;
   _BOOL[221] := FALSE;
   _BOOL[222] := FALSE;
   _BOOL[223] := FALSE;
   _BOOL[224] := FALSE;
   _BOOL[225] := FALSE;
   _BOOL[226] := FALSE;
   _BOOL[227] := FALSE;
   _BOOL[228] := FALSE;
   _BOOL[229] := FALSE;
   _BOOL[230] := FALSE;
   _BOOL[231] := FALSE;
   _BOOL[232] := FALSE;
   _BOOL[233] := FALSE;
   _BOOL[234] := FALSE;
   _BOOL[235] := FALSE;
   _BOOL[236] := FALSE;
   _BOOL[237] := FALSE;
   _BOOL[238] := FALSE;
   _BOOL[239] := FALSE;
   _BOOL[240] := FALSE;
   _BOOL[241] := FALSE;
   _BOOL[242] := FALSE;
   _BOOL[243] := FALSE;
   _BOOL[244] := FALSE;
   _BOOL[245] := FALSE;
   _BOOL[246] := FALSE;
   _BOOL[247] := FALSE;
   _BOOL[248] := FALSE;
   _BOOL[249] := FALSE;
   _BOOL[250] := FALSE;
   _BOOL[251] := FALSE;
   _BOOL[252] := FALSE;
   _BOOL[253] := FALSE;
   _BOOL[254] := FALSE;
   _BOOL[255] := FALSE;
   _BOOL[256] := FALSE;
   _BOOL[257] := FALSE;
   _BOOL[258] := FALSE;
   _BOOL[259] := FALSE;
   _BOOL[260] := FALSE;
   _BOOL[261] := FALSE;
   _BOOL[262] := FALSE;
   _BOOL[263] := FALSE;
   _BOOL[264] := FALSE;
   _BOOL[265] := FALSE;
   _BOOL[266] := FALSE;
   _BOOL[267] := FALSE;
   _BOOL[268] := FALSE;
   _BOOL[269] := FALSE;
   _BOOL[270] := FALSE;
   _BOOL[271] := FALSE;
   _BOOL[272] := FALSE;
   _BOOL[273] := FALSE;
   _BOOL[274] := FALSE;
   _BOOL[275] := FALSE;
   _BOOL[276] := FALSE;
   _BOOL[277] := FALSE;
   _BOOL[278] := FALSE;
   _BOOL[279] := FALSE;
   _BOOL[280] := FALSE;
   _BOOL[281] := FALSE;
   _BOOL[282] := FALSE;
   _BOOL[283] := FALSE;
   _BOOL[284] := FALSE;
   _BOOL[285] := FALSE;
   _BOOL[286] := FALSE;
   _BOOL[287] := FALSE;
   _BOOL[288] := FALSE;
   _BOOL[289] := FALSE;
   _BOOL[290] := FALSE;
   _BOOL[291] := FALSE;
   _BOOL[292] := FALSE;
   _BOOL[293] := FALSE;
   _BOOL[294] := FALSE;
   _BOOL[295] := FALSE;
   _BOOL[296] := FALSE;
   _BOOL[297] := FALSE;
   _BOOL[298] := FALSE;
   _BOOL[299] := FALSE;
   _BOOL[300] := FALSE;
   _BOOL[301] := FALSE;
   _BOOL[302] := FALSE;
   _BOOL[303] := FALSE;
   _BOOL[304] := FALSE;
   _BOOL[305] := FALSE;
   _BOOL[306] := FALSE;
   _BOOL[307] := FALSE;
   _BOOL[308] := FALSE;
   _BOOL[309] := FALSE;
   _BOOL[310] := FALSE;
   _BOOL[311] := FALSE;
   _BOOL[312] := FALSE;
   _BOOL[313] := FALSE;
   _BOOL[314] := FALSE;
   _BOOL[315] := FALSE;
   _BOOL[316] := FALSE;
   _BOOL[317] := FALSE;
   _BOOL[318] := FALSE;
   _BOOL[319] := FALSE;
   _BOOL[320] := FALSE;
   _BOOL[321] := FALSE;
   _BOOL[322] := FALSE;
   _BOOL[323] := FALSE;
   _BOOL[324] := FALSE;
   _BOOL[325] := FALSE;
   _BOOL[326] := FALSE;
   _BOOL[327] := FALSE;
   _BOOL[328] := FALSE;
   _BOOL[329] := FALSE;
   _BOOL[330] := FALSE;
   _BOOL[331] := FALSE;
   _BOOL[332] := FALSE;
   _BOOL[333] := FALSE;
   _BOOL[334] := FALSE;
   _BOOL[335] := FALSE;
   _BOOL[336] := FALSE;
   _BOOL[337] := FALSE;
   _BOOL[338] := FALSE;
   _BOOL[339] := FALSE;
   _BOOL[340] := FALSE;
   _BOOL[341] := FALSE;
   _BOOL[342] := FALSE;
   _BOOL[343] := FALSE;
   _BOOL[344] := FALSE;
   _BOOL[345] := FALSE;
   _BOOL[346] := FALSE;
   _BOOL[347] := FALSE;
   _BOOL[348] := FALSE;
   _BOOL[349] := FALSE;
   _BOOL[350] := FALSE;
   _BOOL[351] := FALSE;
   _BOOL[352] := FALSE;
   _BOOL[353] := FALSE;
   _BOOL[354] := FALSE;
   _BOOL[355] := FALSE;
   _BOOL[356] := FALSE;
   _BOOL[357] := FALSE;
   _BOOL[358] := FALSE;
   _BOOL[359] := FALSE;
   _BOOL[360] := FALSE;
   _BOOL[361] := FALSE;
   _BOOL[362] := FALSE;
   _BOOL[363] := FALSE;
   _BOOL[364] := FALSE;
   _BOOL[365] := FALSE;
   _BOOL[366] := FALSE;
   _BOOL[367] := FALSE;
   _BOOL[368] := FALSE;
   _BOOL[369] := FALSE;
   _BOOL[370] := FALSE;
   _BOOL[371] := FALSE;
   _BOOL[372] := FALSE;
   _BOOL[373] := FALSE;
   _BOOL[374] := FALSE;
   _BOOL[375] := FALSE;
   _BOOL[376] := FALSE;
   _BOOL[377] := FALSE;
   _BOOL[378] := FALSE;
   _BOOL[379] := FALSE;
   _BOOL[380] := FALSE;
   _BOOL[381] := FALSE;
   _BOOL[382] := FALSE;
   _BOOL[383] := FALSE;
   _BOOL[384] := FALSE;
   _BOOL[385] := FALSE;
   _BOOL[386] := FALSE;
   _BOOL[387] := FALSE;
   _BOOL[388] := FALSE;
   _BOOL[389] := FALSE;
   _BOOL[390] := FALSE;
   _BOOL[391] := FALSE;
   _BOOL[392] := FALSE;
   _BOOL[393] := FALSE;
   _BOOL[394] := FALSE;
   _BOOL[395] := FALSE;
   _BOOL[396] := FALSE;
   _BOOL[397] := FALSE;
   _BOOL[398] := FALSE;
   _BOOL[399] := FALSE;
   _BOOL[400] := FALSE;
   _BOOL[401] := FALSE;
   _BOOL[402] := FALSE;
   _BOOL[403] := FALSE;
   _BOOL[404] := FALSE;
   _BOOL[405] := FALSE;
   _BOOL[406] := FALSE;
   _BOOL[407] := FALSE;
   _BOOL[408] := FALSE;
   _BOOL[409] := FALSE;
   _BOOL[410] := FALSE;
   _BOOL[411] := FALSE;
   _BOOL[412] := FALSE;
   _BOOL[413] := FALSE;
   _BOOL[414] := FALSE;
   _BOOL[415] := FALSE;
   _BOOL[416] := FALSE;
   _BOOL[417] := FALSE;
   _BOOL[418] := FALSE;
   _BOOL[419] := FALSE;
   _BOOL[420] := FALSE;
   _BOOL[421] := FALSE;
   _BOOL[422] := FALSE;
   _BOOL[423] := FALSE;
   _BOOL[424] := FALSE;
   _BOOL[425] := FALSE;
   _BOOL[426] := FALSE;
   _BOOL[427] := FALSE;
   _BOOL[428] := FALSE;
   _BOOL[429] := FALSE;
   _BOOL[430] := FALSE;
   _BOOL[431] := FALSE;
   _BOOL[432] := FALSE;
   _BOOL[433] := FALSE;
   _BOOL[434] := FALSE;
   _BOOL[435] := FALSE;
   _BOOL[436] := FALSE;
   _BOOL[437] := FALSE;
   _BOOL[438] := FALSE;
   _BOOL[439] := FALSE;
   _BOOL[440] := FALSE;
   _BOOL[441] := FALSE;
   _BOOL[442] := FALSE;
   _BOOL[443] := FALSE;
   _BOOL[444] := FALSE;
   _BOOL[445] := FALSE;
   _BOOL[446] := FALSE;
   _BOOL[447] := FALSE;
   _BOOL[448] := FALSE;
   _BOOL[449] := FALSE;
   _BOOL[450] := FALSE;
   _BOOL[451] := FALSE;
   _BOOL[452] := FALSE;
   _BOOL[453] := FALSE;
   _BOOL[454] := FALSE;
   _BOOL[455] := FALSE;
   _BOOL[456] := FALSE;
   _BOOL[457] := FALSE;
   _BOOL[458] := FALSE;
   _BOOL[459] := FALSE;
   _BOOL[460] := FALSE;
   _BOOL[461] := FALSE;
   _BOOL[462] := FALSE;
   _BOOL[463] := FALSE;
   _BOOL[464] := FALSE;
   _BOOL[465] := FALSE;
   _BOOL[466] := FALSE;
   _BOOL[467] := FALSE;
   _BOOL[468] := FALSE;
   _BOOL[469] := FALSE;
   _BOOL[470] := FALSE;
   _BOOL[471] := FALSE;
   _BOOL[472] := FALSE;
   _BOOL[473] := FALSE;
   _BOOL[474] := FALSE;
   _BOOL[475] := FALSE;
   _BOOL[476] := FALSE;
   _BOOL[477] := FALSE;
   _BOOL[478] := FALSE;
   _BOOL[479] := FALSE;
   _BOOL[480] := FALSE;
   _BOOL[481] := FALSE;
   _BOOL[482] := FALSE;
   _BOOL[483] := FALSE;
   _BOOL[484] := FALSE;
   _BOOL[485] := FALSE;
   _BOOL[486] := FALSE;
   _BOOL[487] := FALSE;
   _BOOL[488] := FALSE;
   _BOOL[489] := FALSE;
   _BOOL[490] := FALSE;
   _BOOL[491] := FALSE;
   _BOOL[492] := FALSE;
   _BOOL[493] := FALSE;
   _BOOL[494] := FALSE;
   _BOOL[495] := FALSE;
   _BOOL[496] := FALSE;
   _BOOL[497] := FALSE;
   _BOOL[498] := FALSE;
   _BOOL[499] := FALSE;
   _BOOL[500] := FALSE;
   _BOOL[501] := FALSE;
   _BOOL[502] := FALSE;
   _BOOL[503] := FALSE;
   _BOOL[504] := FALSE;
   _BOOL[505] := FALSE;
   _BOOL[506] := FALSE;
   _BOOL[507] := FALSE;
   _BOOL[508] := FALSE;
   _BOOL[509] := FALSE;
   _BOOL[510] := FALSE;
   _BOOL[511] := FALSE;
   _BOOL[512] := FALSE;
END_DATA_BLOCK

DATA_BLOCK "_2015PU040M01_AD"   // DB441
{ S7_Optimized_Access := 'FALSE' }
AUTHOR : FLSmidth
FAMILY : IUSYS
NAME : ADAPTOR
VERSION : 5.2
// stored: InstanceOfName IUSYS_3UF70_V5_MOTOR
"IUSYS_3UF70_V5_MOTOR"
BEGIN
END_DATA_BLOCK

DATA_BLOCK "_2015PU041M01_AD"   // DB442
{ S7_Optimized_Access := 'FALSE' }
AUTHOR : FLSmidth
FAMILY : IUSYS
NAME : ADAPTOR
VERSION : 5.2
// stored: InstanceOfName IUSYS_3UF70_V5_MOTOR
"IUSYS_3UF70_V5_MOTOR"
BEGIN
END_DATA_BLOCK

DATA_BLOCK "IUSYS_INVT_PN_MOTOR_DB"   // DB455
{ S7_Optimized_Access := 'FALSE' }
VERSION : 0.1
// stored: InstanceOfName IUSYS_INVT_PN_MOTOR
"IUSYS_INVT_PN_MOTOR"
BEGIN
END_DATA_BLOCK

DATA_BLOCK "IUSYS_ALTIVAR_PN_MOTOR_TSTR_DB"   // DB462
{ S7_Optimized_Access := 'FALSE' }
VERSION : 0.1
// stored: InstanceOfName IUSYS_ALTIVAR_PN_MOTOR_TSTR
"IUSYS_ALTIVAR_PN_MOTOR_TSTR"
BEGIN
END_DATA_BLOCK

DATA_BLOCK "CIP_COM_CRL_DB"   // DB771
{ S7_Optimized_Access := 'TRUE' }
VERSION : 0.1
// stored: InstanceOfName CIP_COM_CRL
"CIP_COM_CRL"
BEGIN
   T1 := T#10S;
END_DATA_BLOCK

DATA_BLOCK "_997MS100_DB"   // DB1000
TITLE = Instance DB Master: _997MS100
{ S7_Optimized_Access := 'FALSE' }
AUTHOR : METIS
NAME : MAST_DB
VERSION : 8.0
// stored: InstanceOfName ACESYS_MASTER
"ACESYS_MASTER"
BEGIN
   SS_Field_ENABLE := FALSE;
   RED_ENABLE := TRUE;
   WatchDog_HMI_Enable := TRUE;
   WatchDog_HMI_Time := T#30S;
   OB1_CycleTime := 61;
   WatchDog_HMI_Elap := T#6S_558MS;
   MASTER_Link.Flash_Slow := TRUE;
   MASTER_Link.Flash_Fast := TRUE;
   MASTER_Link.SS_FP_Enable := TRUE;
   MASTER_Link.Man_Enable := TRUE;
   MASTER_Link.Loc_Enable := TRUE;
   MASTER_Link.Test_Enable := TRUE;
   MASTER_Link.TimeStamp := 16#B0A8;
   MASTER_Link.OB1_CycleTime := 61;
   BlockInfo.Ace_Version := 80;
   BlockInfo.Ace_BuildNo := 1;
   BlockInfo.DB_Number := 1000;
   Timer_Watchdog.ST := T#13D_5H_8M_51S_558MS;
   Timer_Watchdog.PT := T#30S;
   Timer_Watchdog.RU := TRUE;
   Timer_Watchdog.IN := TRUE;
   TimerSlow_On.ST := T#13D_5H_8M_57S_621MS;
   TimerSlow_On.PT := T#400MS;
   TimerSlow_Off.ST := T#13D_5H_8M_58S_116MS;
   TimerSlow_Off.PT := T#400MS;
   TimerSlow_Off.RU := TRUE;
   TimerSlow_Off.IN := TRUE;
   TimerFast_On.ST := T#13D_5H_8M_57S_868MS;
   TimerFast_On.PT := T#200MS;
   TimerFast_On.IN := TRUE;
   TimerFast_Off.ST := T#13D_5H_8M_57S_560MS;
   TimerFast_Off.PT := T#200MS;
   Flash_Slow := TRUE;
   Flash_Fast := TRUE;
   FirstScan_Hlp := TRUE;
   Clock_Sec_Old := 32;
   Clock_Min_Old := 17;
   Clock_Hour_Old := 5;
   Clock_Day_Old := 22;
   Clock_Month_Old := 6;
   Clock_Year_Old := 2024;
END_DATA_BLOCK

DATA_BLOCK "_997CS100D01_DB"   // DB1001
TITLE = Instance DB Department: _997CS100D01
{ S7_Optimized_Access := 'FALSE' }
AUTHOR : METIS
NAME : DEPT_DB
VERSION : 8.0
// stored: InstanceOfName ACESYS_DEPT
"ACESYS_DEPT"
BEGIN
   Master_Link.Flash_Slow := TRUE;
   Master_Link.Flash_Fast := TRUE;
   Master_Link.SS_FP_Enable := TRUE;
   Master_Link.Man_Enable := TRUE;
   Master_Link.Loc_Enable := TRUE;
   Master_Link.Test_Enable := TRUE;
   Master_Link.TimeStamp := 16#B0AE;
   Master_Link.OB1_CycleTime := 62;
   EnCtrl := TRUE;
   DEMER := TRUE;
   STOP := TRUE;
   DEPT_LINK.TimeStamp := 16#B0AE;
   DEPT_LINK.OB1_CycleTime := 62;
   DEPT_LINK.Flash_Slow := TRUE;
   DEPT_LINK.Flash_Fast := TRUE;
   DEPT_LINK.Man_Enable := TRUE;
   DEPT_LINK.Loc_Enable := TRUE;
   DEPT_LINK.Test_Enable := TRUE;
   DEPT_LINK.SS_FP_Enable := TRUE;
   DEPT_LINK.EmergencyStop := TRUE;
   DEPT_LINK.All_Group_Sel_RDY := TRUE;
   DEPT_LINK.All_Selected_Running := TRUE;
   DEPT_LINK.Ready_For_StopCmd := TRUE;
   MSW.EXT.Operation := TRUE;
   MSW.Status := 14082;
   MSW.TimeStamp := 16#3D5E;
   BlockInfo.Ace_Version := 80;
   BlockInfo.Ace_BuildNo := 1;
   BlockInfo.DB_Number := 1001;
   FP_DIM.Select := TRUE;
   FP_DIM.DeSelect := TRUE;
   FP_DIM.Stop := TRUE;
   FP_DIM.QuickStop := TRUE;
   FP_DIM.MasterStop := TRUE;
   ONS_FS_Reset := TRUE;
   MSW_Status := 14082;
   StatusToECS := 2;
   Dept_Link_Internal.TimeStamp := 16#B0AE;
   Dept_Link_Internal.OB1_CycleTime := 62;
   Dept_Link_Internal.Flash_Slow := TRUE;
   Dept_Link_Internal.Flash_Fast := TRUE;
   Dept_Link_Internal.Man_Enable := TRUE;
   Dept_Link_Internal.Loc_Enable := TRUE;
   Dept_Link_Internal.Test_Enable := TRUE;
   Dept_Link_Internal.SS_FP_Enable := TRUE;
   Dept_Link_Internal.EmergencyStop := TRUE;
   Dept_Link_Internal.All_Group_ON := TRUE;
   Dept_Link_Internal.All_Group_OFF := TRUE;
   Dept_Link_Internal.All_Group_Sel_RDY := TRUE;
   Dept_Link_Internal.All_Selected := TRUE;
   Dept_Link_Internal.All_DeSelected := TRUE;
   Dept_Link_Internal.All_Selected_Running := TRUE;
   MSW_Status_Trans := 14082;
END_DATA_BLOCK

DATA_BLOCK "_995CS100_DEPT01_DB"   // DB1002
TITLE = Instance DB Department: _997CS100_DEPT01
{ S7_Optimized_Access := 'FALSE' }
AUTHOR : METIS
NAME : DEPT_DB
VERSION : 8.0
// stored: InstanceOfName ACESYS_DEPT
"ACESYS_DEPT"
BEGIN
END_DATA_BLOCK

DATA_BLOCK "_997CD100G01_DB"   // DB1500
TITLE = Instance DB Group: _997CD100G01
{ S7_Optimized_Access := 'FALSE' }
AUTHOR : METIS
NAME : GROUP_DB
VERSION : 8.0
// stored: InstanceOfName ACESYS_GROUP
"ACESYS_GROUP"
BEGIN
   FP_SEL.DeptCtrl := TRUE;
   FP_PARM.StartWarn_Pre := 15;
   FP_PARM.StartFail_Pre := 120;
   FP_PARM.StopFail_Pre := 120;
   EnCtrl := TRUE;
   INTL.OK := TRUE;
   INTL.DetectFirst := TRUE;
   INTL.ClearFirst := TRUE;
   INTL_SEQ_STR.OK := TRUE;
   INTL_SEQ_STR.DetectFirst := TRUE;
   INTL_SEQ_STR.ClearFirst := TRUE;
   INTL_SEQ_STP.OK := TRUE;
   RDY_START := TRUE;
   GRP_OFF := TRUE;
   TOKEN.TimeStamp := 16#B0B5;
   TOKEN.OB1_CycleTime := 62;
   TOKEN.AL_UNIT := TRUE;
   TOKEN.GON := TRUE;
   TOKEN.GOFF := TRUE;
   TOKEN.Interlock_Unit := TRUE;
   TOKEN.Flash_Slow := TRUE;
   TOKEN.Flash_Fast := TRUE;
   TOKEN.EmergencyStop := TRUE;
   TOKEN.SS_FP_Enable := TRUE;
   TOKEN.Man_Enable := TRUE;
   TOKEN.Loc_Enable := TRUE;
   TOKEN.TEST_Enable := TRUE;
   TOKEN.AllUnitsAuto := TRUE;
   TOKEN.ResetNotEmpty := TRUE;
   TOKEN.AlarmSuppres := TRUE;
   TOKEN.SACK_On := TRUE;
   TOKEN.SACK_Off := TRUE;
   MSW.Status := 8193;
   MSW.TimeStamp := 16#5FEF;
   BlockInfo.Ace_Version := 80;
   BlockInfo.Ace_BuildNo := 4;
   BlockInfo.State_Act := 101;
   BlockInfo.State_Prev := 190;
   BlockInfo.DB_Number := 1500;
   FP_CMD.Auto := TRUE;
   FP_DIM.Select := TRUE;
   FP_DIM.Local := TRUE;
   FP_DIM.SS_FP := TRUE;
   FP_SHOW.Auto := TRUE;
   FP_SHOW.Local := TRUE;
   FP_SHOW.SS_FP := TRUE;
   FP_PARM.StartWarn_Acc := 15;
   FP_PARM.StartFail_Acc := 120;
   FP_PARM.StopFail_Acc := 120;
   FP_PARM.StopReason := 99;
   FP_PARM.INTL := TRUE;
   FP_PARM.INTL_SEQ_STR := TRUE;
   FP_PARM.INTL_SEQ_STP := TRUE;
   STATE.Stopped := TRUE;
   ONS.Cmd_Auto := TRUE;
   ONS.Pause := TRUE;
   ONS.SecPulse2 := TRUE;
   StartWarn_Mem := 15;
   StartFail_Mem := 120;
   StopFail_Mem := 120;
   ModePointer := 51;
   StatusWork := 1;
   ECSStatusBuilder := 8192;
   MSW_Status := 8193;
   ModeAuto := TRUE;
   RST_TMR.ST := T#13D_3H_58M_51S_335MS;
   RST_TMR.PT := T#1S;
   OUT.RDY_START := TRUE;
   OUT.GRP_OFF := TRUE;
   OUT.INTL_OK_STAT := TRUE;
   OUT.INTL_SEQ_STR_OK_STAT := TRUE;
   OUT.INTL_SEQ_STP_OK_STAT := TRUE;
   TOKEN_Stat.TimeStamp := 16#B0B5;
   TOKEN_Stat.OB1_CycleTime := 62;
   TOKEN_Stat.AL_UNIT := TRUE;
   TOKEN_Stat.GON := TRUE;
   TOKEN_Stat.GOFF := TRUE;
   TOKEN_Stat.Interlock_Unit := TRUE;
   TOKEN_Stat.Flash_Slow := TRUE;
   TOKEN_Stat.Flash_Fast := TRUE;
   TOKEN_Stat.EmergencyStop := TRUE;
   TOKEN_Stat.SS_FP_Enable := TRUE;
   TOKEN_Stat.Man_Enable := TRUE;
   TOKEN_Stat.Loc_Enable := TRUE;
   TOKEN_Stat.TEST_Enable := TRUE;
   TOKEN_Stat.AllUnitsAuto := TRUE;
   TOKEN_Stat.ResetNotEmpty := TRUE;
   TOKEN_Stat.AlarmSuppres := TRUE;
   TOKEN_Stat.SACK_On := TRUE;
   TOKEN_Stat.SACK_Off := TRUE;
   MSW_Status_Trans := 8193;
END_DATA_BLOCK

DATA_BLOCK "_997CD100G02_DB"   // DB1501
TITLE = Instance DB Group: _997CD100G02
{ S7_Optimized_Access := 'FALSE' }
AUTHOR : METIS
NAME : GROUP_DB
VERSION : 8.0
// stored: InstanceOfName ACESYS_GROUP
"ACESYS_GROUP"
BEGIN
   FP_SEL.DeptCtrl := TRUE;
   FP_PARM.StartWarn_Pre := 1;
   FP_PARM.StartFail_Pre := 120;
   FP_PARM.StopFail_Pre := 120;
   EnCtrl := TRUE;
   INTL.OK := TRUE;
   INTL.DetectFirst := TRUE;
   INTL.ClearFirst := TRUE;
   INTL_SEQ_STR.OK := TRUE;
   INTL_SEQ_STR.DetectFirst := TRUE;
   INTL_SEQ_STR.ClearFirst := TRUE;
   INTL_SEQ_STP.OK := TRUE;
   RDY_START := TRUE;
   GRP_OFF := TRUE;
   TOKEN.TimeStamp := 16#B0BB;
   TOKEN.OB1_CycleTime := 59;
   TOKEN.AL_UNIT := TRUE;
   TOKEN.GON := TRUE;
   TOKEN.GOFF := TRUE;
   TOKEN.Interlock_Unit := TRUE;
   TOKEN.Flash_Slow := TRUE;
   TOKEN.Flash_Fast := TRUE;
   TOKEN.EmergencyStop := TRUE;
   TOKEN.SS_FP_Enable := TRUE;
   TOKEN.Man_Enable := TRUE;
   TOKEN.Loc_Enable := TRUE;
   TOKEN.TEST_Enable := TRUE;
   TOKEN.AllUnitsAuto := TRUE;
   TOKEN.ResetNotEmpty := TRUE;
   TOKEN.AlarmSuppres := TRUE;
   TOKEN.SACK_On := TRUE;
   TOKEN.SACK_Off := TRUE;
   TOKEN.UnitSelect := TRUE;
   MSW.Status := 8193;
   MSW.TimeStamp := 16#9D0E;
   BlockInfo.Ace_Version := 80;
   BlockInfo.Ace_BuildNo := 4;
   BlockInfo.State_Act := 101;
   BlockInfo.State_Prev := 190;
   BlockInfo.DB_Number := 1501;
   FP_CMD.Auto := TRUE;
   FP_DIM.Select := TRUE;
   FP_DIM.Local := TRUE;
   FP_DIM.SS_FP := TRUE;
   FP_SHOW.Auto := TRUE;
   FP_SHOW.Local := TRUE;
   FP_SHOW.SS_FP := TRUE;
   FP_PARM.StartWarn_Acc := 1;
   FP_PARM.StartFail_Acc := 120;
   FP_PARM.StopFail_Acc := 120;
   FP_PARM.StopReason := 99;
   FP_PARM.INTL := TRUE;
   FP_PARM.INTL_SEQ_STR := TRUE;
   FP_PARM.INTL_SEQ_STP := TRUE;
   STATE.Stopped := TRUE;
   ONS.Cmd_Auto := TRUE;
   ONS.Pause := TRUE;
   ONS.SecPulse2 := TRUE;
   StartWarn_Mem := 1;
   StartFail_Mem := 120;
   StopFail_Mem := 120;
   ModePointer := 51;
   StatusWork := 1;
   ECSStatusBuilder := 8192;
   MSW_Status := 8193;
   ModeAuto := TRUE;
   RST_TMR.ST := T#13D_3H_58M_51S_335MS;
   RST_TMR.PT := T#1S;
   OUT.RDY_START := TRUE;
   OUT.GRP_OFF := TRUE;
   OUT.INTL_OK_STAT := TRUE;
   OUT.INTL_SEQ_STR_OK_STAT := TRUE;
   OUT.INTL_SEQ_STP_OK_STAT := TRUE;
   TOKEN_Stat.TimeStamp := 16#B0BB;
   TOKEN_Stat.OB1_CycleTime := 59;
   TOKEN_Stat.AL_UNIT := TRUE;
   TOKEN_Stat.GON := TRUE;
   TOKEN_Stat.GOFF := TRUE;
   TOKEN_Stat.Interlock_Unit := TRUE;
   TOKEN_Stat.Flash_Slow := TRUE;
   TOKEN_Stat.Flash_Fast := TRUE;
   TOKEN_Stat.EmergencyStop := TRUE;
   TOKEN_Stat.SS_FP_Enable := TRUE;
   TOKEN_Stat.Man_Enable := TRUE;
   TOKEN_Stat.Loc_Enable := TRUE;
   TOKEN_Stat.TEST_Enable := TRUE;
   TOKEN_Stat.AllUnitsAuto := TRUE;
   TOKEN_Stat.ResetNotEmpty := TRUE;
   TOKEN_Stat.AlarmSuppres := TRUE;
   TOKEN_Stat.SACK_On := TRUE;
   TOKEN_Stat.SACK_Off := TRUE;
   MSW_Status_Trans := 8193;
END_DATA_BLOCK

DATA_BLOCK "_997CD100G03_DB"   // DB1502
TITLE = Instance DB Group: _997CD100G03
{ S7_Optimized_Access := 'FALSE' }
AUTHOR : METIS
NAME : GROUP_DB
VERSION : 8.0
// stored: InstanceOfName ACESYS_GROUP
"ACESYS_GROUP"
BEGIN
   FP_SEL.DeptCtrl := TRUE;
   FP_PARM.StartWarn_Pre := 5;
   FP_PARM.StartFail_Pre := 120;
   FP_PARM.StopFail_Pre := 600;
   EnCtrl := TRUE;
   INTL.OK := TRUE;
   INTL.DetectFirst := TRUE;
   INTL.ClearFirst := TRUE;
   INTL_SEQ_STR.OK := TRUE;
   INTL_SEQ_STR.DetectFirst := TRUE;
   INTL_SEQ_STR.ClearFirst := TRUE;
   INTL_SEQ_STP.OK := TRUE;
   GSEL := TRUE;
   GACC := TRUE;
   GRUN := TRUE;
   RDY_START := TRUE;
   CMD_OUT.GSEL := TRUE;
   TOKEN.TimeStamp := 16#B0BB;
   TOKEN.OB1_CycleTime := 59;
   TOKEN.AL_UNIT := TRUE;
   TOKEN.GON := TRUE;
   TOKEN.Interlock_Unit := TRUE;
   TOKEN.Flash_Slow := TRUE;
   TOKEN.Flash_Fast := TRUE;
   TOKEN.EmergencyStop := TRUE;
   TOKEN.SS_FP_Enable := TRUE;
   TOKEN.Man_Enable := TRUE;
   TOKEN.Loc_Enable := TRUE;
   TOKEN.TEST_Enable := TRUE;
   TOKEN.AllUnitsAuto := TRUE;
   TOKEN.ResetNotEmpty := TRUE;
   TOKEN.SACK_On := TRUE;
   TOKEN.UnitSelect := TRUE;
   MSW.EXT.Operation := TRUE;
   MSW.Status := 4104;
   MSW.TimeStamp := 16#3D5B;
   BlockInfo.Ace_Version := 80;
   BlockInfo.Ace_BuildNo := 4;
   BlockInfo.State_Act := 108;
   BlockInfo.State_Prev := 106;
   BlockInfo.DB_Number := 1502;
   FP_CMD.Auto := TRUE;
   FP_DIM.Deselect := TRUE;
   FP_DIM.SS_FP := TRUE;
   FP_SHOW.Auto := TRUE;
   FP_SHOW.Local := TRUE;
   FP_SHOW.SS_FP := TRUE;
   FP_PARM.StartWarn_Acc := 5;
   FP_PARM.StartFail_Acc := 120;
   FP_PARM.StopFail_Acc := 600;
   FP_PARM.INTL := TRUE;
   FP_PARM.INTL_SEQ_STR := TRUE;
   FP_PARM.INTL_SEQ_STP := TRUE;
   STATE.Running := TRUE;
   ONS.Cmd_Auto := TRUE;
   ONS.Pause := TRUE;
   ONS.SecPulse2 := TRUE;
   StartWarn_Mem := 5;
   StartFail_Mem := 120;
   StopFail_Mem := 600;
   ModePointer := 51;
   StatusWork := 8;
   ECSStatusBuilder := 4096;
   MSW_Status := 4104;
   ModeAuto := TRUE;
   RST_TMR.ST := T#13D_3H_58M_51S_340MS;
   RST_TMR.PT := T#1S;
   OUT.GSEL := TRUE;
   OUT.GACC := TRUE;
   OUT.GRUN := TRUE;
   OUT.RDY_START := TRUE;
   OUT.INTL_OK_STAT := TRUE;
   OUT.INTL_SEQ_STR_OK_STAT := TRUE;
   OUT.INTL_SEQ_STP_OK_STAT := TRUE;
   TOKEN_Stat.TimeStamp := 16#B0BB;
   TOKEN_Stat.OB1_CycleTime := 59;
   TOKEN_Stat.AL_UNIT := TRUE;
   TOKEN_Stat.GON := TRUE;
   TOKEN_Stat.Interlock_Unit := TRUE;
   TOKEN_Stat.Flash_Slow := TRUE;
   TOKEN_Stat.Flash_Fast := TRUE;
   TOKEN_Stat.EmergencyStop := TRUE;
   TOKEN_Stat.SS_FP_Enable := TRUE;
   TOKEN_Stat.Man_Enable := TRUE;
   TOKEN_Stat.Loc_Enable := TRUE;
   TOKEN_Stat.TEST_Enable := TRUE;
   TOKEN_Stat.AllUnitsAuto := TRUE;
   TOKEN_Stat.ResetNotEmpty := TRUE;
   TOKEN_Stat.SACK_On := TRUE;
   TOKEN_Stat.SACK_Off := TRUE;
   MSW_Status_Trans := 4104;
END_DATA_BLOCK

DATA_BLOCK "_997CD100G04_DB"   // DB1503
TITLE = Instance DB Group: _997CD100G04
{ S7_Optimized_Access := 'FALSE' }
AUTHOR : METIS
NAME : GROUP_DB
VERSION : 8.0
// stored: InstanceOfName ACESYS_GROUP
"ACESYS_GROUP"
BEGIN
   FP_SEL.DeptCtrl := TRUE;
   FP_PARM.StartWarn_Pre := 15;
   FP_PARM.StartFail_Pre := 120;
   FP_PARM.StopFail_Pre := 120;
   EnCtrl := TRUE;
   GON := FALSE;
   GOFF := FALSE;
   INTL.OK := TRUE;
   INTL_SEQ_STR.OK := TRUE;
   INTL_SEQ_STP.OK := TRUE;
   RDY_START := TRUE;
   TOKEN.TimeStamp := 16#B0BB;
   TOKEN.OB1_CycleTime := 59;
   TOKEN.AL_UNIT := TRUE;
   TOKEN.Interlock_Unit := TRUE;
   TOKEN.Flash_Slow := TRUE;
   TOKEN.Flash_Fast := TRUE;
   TOKEN.EmergencyStop := TRUE;
   TOKEN.SS_FP_Enable := TRUE;
   TOKEN.Man_Enable := TRUE;
   TOKEN.Loc_Enable := TRUE;
   TOKEN.TEST_Enable := TRUE;
   TOKEN.AllUnitsAuto := TRUE;
   TOKEN.ResetNotEmpty := TRUE;
   TOKEN.SACK_On := TRUE;
   TOKEN.SACK_Off := TRUE;
   MSW.Status := 8215;
   MSW.TimeStamp := 16#5FEF;
   BlockInfo.Ace_Version := 80;
   BlockInfo.Ace_BuildNo := 4;
   BlockInfo.State_Act := 101;
   BlockInfo.State_Prev := 103;
   BlockInfo.DB_Number := 1503;
   FP_CMD.Auto := TRUE;
   FP_DIM.Select := TRUE;
   FP_DIM.Local := TRUE;
   FP_DIM.SS_FP := TRUE;
   FP_SHOW.Auto := TRUE;
   FP_SHOW.Local := TRUE;
   FP_SHOW.SS_FP := TRUE;
   FP_PARM.StartWarn_Acc := 15;
   FP_PARM.StartFail_Acc := 120;
   FP_PARM.StopFail_Acc := 120;
   FP_PARM.StopReason := 10;
   FP_PARM.INTL := TRUE;
   FP_PARM.INTL_SEQ_STR := TRUE;
   FP_PARM.INTL_SEQ_STP := TRUE;
   STATE.Stopped := TRUE;
   ONS.Cmd_Auto := TRUE;
   ONS.Pause := TRUE;
   ONS.SecPulse2 := TRUE;
   StartWarn_Mem := 15;
   StartFail_Mem := 120;
   StopFail_Mem := 120;
   ModePointer := 51;
   StatusWork := 23;
   ECSStatusBuilder := 8192;
   MSW_Status := 8215;
   ModeAuto := TRUE;
   RST_TMR.ST := T#13D_3H_58M_51S_352MS;
   RST_TMR.PT := T#1S;
   OUT.RDY_START := TRUE;
   OUT.INTL_OK_STAT := TRUE;
   OUT.INTL_SEQ_STR_OK_STAT := TRUE;
   OUT.INTL_SEQ_STP_OK_STAT := TRUE;
   TOKEN_Stat.TimeStamp := 16#B0BB;
   TOKEN_Stat.OB1_CycleTime := 59;
   TOKEN_Stat.AL_UNIT := TRUE;
   TOKEN_Stat.Interlock_Unit := TRUE;
   TOKEN_Stat.Flash_Slow := TRUE;
   TOKEN_Stat.Flash_Fast := TRUE;
   TOKEN_Stat.EmergencyStop := TRUE;
   TOKEN_Stat.SS_FP_Enable := TRUE;
   TOKEN_Stat.Man_Enable := TRUE;
   TOKEN_Stat.Loc_Enable := TRUE;
   TOKEN_Stat.TEST_Enable := TRUE;
   TOKEN_Stat.AllUnitsAuto := TRUE;
   TOKEN_Stat.ResetNotEmpty := TRUE;
   TOKEN_Stat.SACK_On := TRUE;
   TOKEN_Stat.SACK_Off := TRUE;
   MSW_Status_Trans := 8215;
END_DATA_BLOCK

DATA_BLOCK "_995CD100G50_DB"   // DB1550
{ S7_Optimized_Access := 'FALSE' }
AUTHOR : FLSmidth
FAMILY : ACESYS
NAME : GROUP
VERSION : 8.0
// stored: InstanceOfName ACESYS_GROUP
"ACESYS_GROUP"
BEGIN
END_DATA_BLOCK

DATA_BLOCK "_2010CV300D20Z43_DB"   // DB2000
TITLE = Instance DB Alarm:
{ S7_Optimized_Access := 'FALSE' }
AUTHOR : METIS
NAME : ALARM_DB
VERSION : 8.0
// stored: InstanceOfName ACESYS_ALARM
"ACESYS_ALARM"
BEGIN
   FP_EN.Alarm_Low := TRUE;
   PWR := TRUE;
   EN_L := TRUE;
   OK := TRUE;
   AL_L := TRUE;
   AL_H := TRUE;
   WARN_L := TRUE;
   WARN_H := TRUE;
   MSW.EXT.Operation := TRUE;
   MSW.Status := 2;
   MSW.TimeStamp := 16#2B0B;
   BlockInfo.Ace_Version := 80;
   BlockInfo.Ace_BuildNo := 4;
   BlockInfo.State_Act := 2;
   BlockInfo.State_Prev := 202;
   BlockInfo.DB_Number := 2000;
   FP_SIM.SIG_Enable := TRUE;
   FP_SIM.PWR_Enable := TRUE;
   ONS.SecPulse2 := TRUE;
   ONS.AL_L_Aux := TRUE;
   ONS.AL_H_Aux := TRUE;
   EnableTime_Low_Done := TRUE;
   StatusWork := 2;
   OUT.OK := TRUE;
   OUT.AL_L := TRUE;
   OUT.AL_H := TRUE;
   OUT.WARN_L := TRUE;
   OUT.WARN_H := TRUE;
   MSW_Status_Trans := 2;
END_DATA_BLOCK

DATA_BLOCK "_2010CV300D19Z43_DB"   // DB2001
TITLE = Instance DB Alarm:
{ S7_Optimized_Access := 'FALSE' }
AUTHOR : METIS
NAME : ALARM_DB
VERSION : 8.0
// stored: InstanceOfName ACESYS_ALARM
"ACESYS_ALARM"
BEGIN
   FP_EN.Alarm_Low := TRUE;
   PWR := TRUE;
   EN_L := TRUE;
   OK := TRUE;
   AL_L := TRUE;
   AL_H := TRUE;
   WARN_L := TRUE;
   WARN_H := TRUE;
   MSW.EXT.Operation := TRUE;
   MSW.Status := 2;
   MSW.TimeStamp := 16#531C;
   BlockInfo.Ace_Version := 80;
   BlockInfo.Ace_BuildNo := 4;
   BlockInfo.State_Act := 2;
   BlockInfo.State_Prev := 202;
   BlockInfo.DB_Number := 2001;
   FP_SIM.SIG_Enable := TRUE;
   FP_SIM.PWR_Enable := TRUE;
   ONS.SecPulse2 := TRUE;
   ONS.AL_L_Aux := TRUE;
   ONS.AL_H_Aux := TRUE;
   EnableTime_Low_Done := TRUE;
   StatusWork := 2;
   OUT.OK := TRUE;
   OUT.AL_L := TRUE;
   OUT.AL_H := TRUE;
   OUT.WARN_L := TRUE;
   OUT.WARN_H := TRUE;
   MSW_Status_Trans := 2;
END_DATA_BLOCK

DATA_BLOCK "_2010CV300D06Z41_DB"   // DB2002
TITLE = Instance DB Alarm:
{ S7_Optimized_Access := 'FALSE' }
AUTHOR : METIS
NAME : ALARM_DB
VERSION : 8.0
// stored: InstanceOfName ACESYS_ALARM
"ACESYS_ALARM"
BEGIN
   FP_PARM.EnableTime_Low_Pre := 5;
   FP_EN.ParentSupress := TRUE;
   FP_EN.ParentSupressUnit := TRUE;
   PWR := TRUE;
   EN_L := TRUE;
   OK := TRUE;
   AL_L := TRUE;
   AL_H := TRUE;
   WARN_L := TRUE;
   WARN_H := TRUE;
   MSW.EXT.Operation := TRUE;
   MSW.Status := 2;
   MSW.TimeStamp := 16#9174;
   BlockInfo.Ace_Version := 80;
   BlockInfo.Ace_BuildNo := 4;
   BlockInfo.State_Act := 2;
   BlockInfo.State_Prev := 1;
   BlockInfo.DB_Number := 2002;
   FP_PARM.EnableTime_Low_Acc := 5;
   FP_PARM.AlarmDelay_Low_Pre := 7;
   FP_PARM.AlarmDelay_Low_Acc := 7;
   FP_EN.Warning_Low := TRUE;
   FP_SIM.SIG_Enable := TRUE;
   FP_SIM.PWR_Enable := TRUE;
   ONS.SecPulse2 := TRUE;
   ONS.AL_L_Aux := TRUE;
   ONS.AL_H_Aux := TRUE;
   EnableTime_Low_Done := TRUE;
   StatusWork := 2;
   AlarmDelay_Low_Mem := 7;
   OUT.OK := TRUE;
   OUT.AL_L := TRUE;
   OUT.AL_H := TRUE;
   OUT.WARN_L := TRUE;
   OUT.WARN_H := TRUE;
   MSW_Status_Trans := 2;
END_DATA_BLOCK

DATA_BLOCK "_2010CV300D06Z42_DB"   // DB2003
TITLE = Instance DB Alarm:
{ S7_Optimized_Access := 'FALSE' }
AUTHOR : METIS
NAME : ALARM_DB
VERSION : 8.0
// stored: InstanceOfName ACESYS_ALARM
"ACESYS_ALARM"
BEGIN
   FP_PARM.EnableTime_Low_Pre := 5;
   FP_EN.ParentSupress := TRUE;
   FP_EN.ParentSupressUnit := TRUE;
   PWR := TRUE;
   EN_L := TRUE;
   OK := TRUE;
   AL_L := TRUE;
   AL_H := TRUE;
   WARN_L := TRUE;
   WARN_H := TRUE;
   MSW.EXT.Operation := TRUE;
   MSW.Status := 2;
   MSW.TimeStamp := 16#43A7;
   BlockInfo.Ace_Version := 80;
   BlockInfo.Ace_BuildNo := 4;
   BlockInfo.State_Act := 2;
   BlockInfo.State_Prev := 1;
   BlockInfo.DB_Number := 2003;
   FP_PARM.EnableTime_Low_Acc := 5;
   FP_EN.Warning_Low := TRUE;
   FP_SIM.SIG_Enable := TRUE;
   FP_SIM.PWR_Enable := TRUE;
   ONS.SecPulse2 := TRUE;
   ONS.AL_L_Aux := TRUE;
   ONS.AL_H_Aux := TRUE;
   EnableTime_Low_Done := TRUE;
   StatusWork := 2;
   OUT.OK := TRUE;
   OUT.AL_L := TRUE;
   OUT.AL_H := TRUE;
   OUT.WARN_L := TRUE;
   OUT.WARN_H := TRUE;
   MSW_Status_Trans := 2;
END_DATA_BLOCK

DATA_BLOCK "_2010CV300D06Z44_DB"   // DB2004
TITLE = Instance DB Alarm:
{ S7_Optimized_Access := 'FALSE' }
AUTHOR : METIS
NAME : ALARM_DB
VERSION : 8.0
// stored: InstanceOfName ACESYS_ALARM
"ACESYS_ALARM"
BEGIN
   FP_PARM.EnableTime_Low_Pre := 1;
   FP_EN.Alarm_Low := TRUE;
   PWR := TRUE;
   EN_L := TRUE;
   OK := TRUE;
   AL_L := TRUE;
   AL_H := TRUE;
   WARN_L := TRUE;
   WARN_H := TRUE;
   MSW.EXT.Operation := TRUE;
   MSW.Status := 2;
   MSW.TimeStamp := 16#92F4;
   BlockInfo.Ace_Version := 80;
   BlockInfo.Ace_BuildNo := 4;
   BlockInfo.State_Act := 2;
   BlockInfo.State_Prev := 1;
   BlockInfo.DB_Number := 2004;
   FP_PARM.EnableTime_Low_Acc := 1;
   FP_SIM.SIG_Enable := TRUE;
   FP_SIM.PWR_Enable := TRUE;
   ONS.SecPulse2 := TRUE;
   ONS.AL_L_Aux := TRUE;
   ONS.AL_H_Aux := TRUE;
   EnableTime_Low_Done := TRUE;
   StatusWork := 2;
   OUT.OK := TRUE;
   OUT.AL_L := TRUE;
   OUT.AL_H := TRUE;
   OUT.WARN_L := TRUE;
   OUT.WARN_H := TRUE;
   MSW_Status_Trans := 2;
END_DATA_BLOCK

DATA_BLOCK "_2010CV300D06Z45_DB"   // DB2005
TITLE = Instance DB Alarm:
{ S7_Optimized_Access := 'FALSE' }
AUTHOR : METIS
NAME : ALARM_DB
VERSION : 8.0
// stored: InstanceOfName ACESYS_ALARM
"ACESYS_ALARM"
BEGIN
   FP_PARM.EnableTime_Low_Pre := 1;
   FP_EN.Alarm_Low := TRUE;
   PWR := TRUE;
   EN_L := TRUE;
   OK := TRUE;
   AL_L := TRUE;
   AL_H := TRUE;
   WARN_L := TRUE;
   WARN_H := TRUE;
   MSW.EXT.Operation := TRUE;
   MSW.Status := 2;
   MSW.TimeStamp := 16#49C7;
   BlockInfo.Ace_Version := 80;
   BlockInfo.Ace_BuildNo := 4;
   BlockInfo.State_Act := 2;
   BlockInfo.State_Prev := 1;
   BlockInfo.DB_Number := 2005;
   FP_PARM.EnableTime_Low_Acc := 1;
   FP_SIM.SIG_Enable := TRUE;
   FP_SIM.PWR_Enable := TRUE;
   ONS.SecPulse2 := TRUE;
   ONS.AL_L_Aux := TRUE;
   ONS.AL_H_Aux := TRUE;
   EnableTime_Low_Done := TRUE;
   StatusWork := 2;
   OUT.OK := TRUE;
   OUT.AL_L := TRUE;
   OUT.AL_H := TRUE;
   OUT.WARN_L := TRUE;
   OUT.WARN_H := TRUE;
   MSW_Status_Trans := 2;
END_DATA_BLOCK

DATA_BLOCK "_2010CV300D06Z46_DB"   // DB2006
TITLE = Instance DB Alarm:
{ S7_Optimized_Access := 'FALSE' }
AUTHOR : METIS
NAME : ALARM_DB
VERSION : 8.0
// stored: InstanceOfName ACESYS_ALARM
"ACESYS_ALARM"
BEGIN
   FP_PARM.EnableTime_Low_Pre := 1;
   FP_EN.Alarm_Low := TRUE;
   PWR := TRUE;
   EN_L := TRUE;
   OK := TRUE;
   AL_L := TRUE;
   AL_H := TRUE;
   WARN_L := TRUE;
   WARN_H := TRUE;
   MSW.EXT.Operation := TRUE;
   MSW.Status := 2;
   MSW.TimeStamp := 16#3034;
   BlockInfo.Ace_Version := 80;
   BlockInfo.Ace_BuildNo := 4;
   BlockInfo.State_Act := 2;
   BlockInfo.State_Prev := 202;
   BlockInfo.DB_Number := 2006;
   FP_PARM.EnableTime_Low_Acc := 1;
   FP_SIM.SIG_Enable := TRUE;
   FP_SIM.PWR_Enable := TRUE;
   ONS.SecPulse2 := TRUE;
   ONS.AL_L_Aux := TRUE;
   ONS.AL_H_Aux := TRUE;
   EnableTime_Low_Done := TRUE;
   StatusWork := 2;
   OUT.OK := TRUE;
   OUT.AL_L := TRUE;
   OUT.AL_H := TRUE;
   OUT.WARN_L := TRUE;
   OUT.WARN_H := TRUE;
   MSW_Status_Trans := 2;
END_DATA_BLOCK

DATA_BLOCK "_2010CV300U01SSW02_DB"   // DB2007
TITLE = Instance DB Alarm:
{ S7_Optimized_Access := 'FALSE' }
AUTHOR : METIS
NAME : ALARM_DB
VERSION : 8.0
// stored: InstanceOfName ACESYS_ALARM
"ACESYS_ALARM"
BEGIN
   FP_EN.Alarm_Low := TRUE;
   PWR := TRUE;
   EN_L := TRUE;
   OK := TRUE;
   AL_L := TRUE;
   AL_H := TRUE;
   WARN_L := TRUE;
   WARN_H := TRUE;
   MSW.EXT.Operation := TRUE;
   MSW.Status := 2;
   MSW.TimeStamp := 16#E560;
   BlockInfo.Ace_Version := 80;
   BlockInfo.Ace_BuildNo := 4;
   BlockInfo.State_Act := 2;
   BlockInfo.State_Prev := 202;
   BlockInfo.DB_Number := 2007;
   FP_SIM.SIG_Enable := TRUE;
   FP_SIM.PWR_Enable := TRUE;
   ONS.SecPulse2 := TRUE;
   ONS.AL_L_Aux := TRUE;
   ONS.AL_H_Aux := TRUE;
   EnableTime_Low_Done := TRUE;
   StatusWork := 2;
   OUT.OK := TRUE;
   OUT.AL_L := TRUE;
   OUT.AL_H := TRUE;
   OUT.WARN_L := TRUE;
   OUT.WARN_H := TRUE;
   MSW_Status_Trans := 2;
END_DATA_BLOCK

DATA_BLOCK "_2010CV300U01SSW03_DB"   // DB2008
TITLE = Instance DB Alarm:
{ S7_Optimized_Access := 'FALSE' }
AUTHOR : METIS
NAME : ALARM_DB
VERSION : 8.0
// stored: InstanceOfName ACESYS_ALARM
"ACESYS_ALARM"
BEGIN
   FP_EN.Alarm_Low := TRUE;
   PWR := TRUE;
   EN_L := TRUE;
   OK := TRUE;
   AL_L := TRUE;
   AL_H := TRUE;
   WARN_L := TRUE;
   WARN_H := TRUE;
   MSW.EXT.Operation := TRUE;
   MSW.Status := 2;
   MSW.TimeStamp := 16#BCB7;
   BlockInfo.Ace_Version := 80;
   BlockInfo.Ace_BuildNo := 4;
   BlockInfo.State_Act := 2;
   BlockInfo.State_Prev := 202;
   BlockInfo.DB_Number := 2008;
   FP_SIM.SIG_Enable := TRUE;
   FP_SIM.PWR_Enable := TRUE;
   ONS.SecPulse2 := TRUE;
   ONS.AL_L_Aux := TRUE;
   ONS.AL_H_Aux := TRUE;
   EnableTime_Low_Done := TRUE;
   StatusWork := 2;
   OUT.OK := TRUE;
   OUT.AL_L := TRUE;
   OUT.AL_H := TRUE;
   OUT.WARN_L := TRUE;
   OUT.WARN_H := TRUE;
   MSW_Status_Trans := 2;
END_DATA_BLOCK

DATA_BLOCK "_2010CV300D01S41_DB"   // DB2009
TITLE = Instance DB Alarm:
{ S7_Optimized_Access := 'FALSE' }
AUTHOR : METIS
NAME : ALARM_DB
VERSION : 8.0
// stored: InstanceOfName ACESYS_ALARM
"ACESYS_ALARM"
BEGIN
   FP_PARM.EnableTime_Low_Pre := 5;
   FP_EN.Alarm_Low := TRUE;
   PWR := TRUE;
   EN_L := TRUE;
   OK := TRUE;
   AL_L := TRUE;
   AL_H := TRUE;
   WARN_L := TRUE;
   WARN_H := TRUE;
   MSW.EXT.Operation := TRUE;
   MSW.Status := 2;
   MSW.TimeStamp := 16#3198;
   BlockInfo.Ace_Version := 80;
   BlockInfo.Ace_BuildNo := 4;
   BlockInfo.State_Act := 2;
   BlockInfo.State_Prev := 1;
   BlockInfo.DB_Number := 2009;
   FP_PARM.EnableTime_Low_Acc := 5;
   FP_SIM.SIG_Enable := TRUE;
   FP_SIM.PWR_Enable := TRUE;
   ONS.SecPulse2 := TRUE;
   ONS.AL_L_Aux := TRUE;
   ONS.AL_H_Aux := TRUE;
   EnableTime_Low_Done := TRUE;
   StatusWork := 2;
   OUT.OK := TRUE;
   OUT.AL_L := TRUE;
   OUT.AL_H := TRUE;
   OUT.WARN_L := TRUE;
   OUT.WARN_H := TRUE;
   MSW_Status_Trans := 2;
END_DATA_BLOCK

DATA_BLOCK "_2010LV100Q02E41_DB"   // DB2010
TITLE = Instance DB Alarm:
{ S7_Optimized_Access := 'FALSE' }
AUTHOR : METIS
NAME : ALARM_DB
VERSION : 8.0
// stored: InstanceOfName ACESYS_ALARM
"ACESYS_ALARM"
BEGIN
   FP_PARM.EnableTime_Low_Pre := 5;
   FP_EN.ParentSupress := TRUE;
   FP_EN.ParentSupressUnit := TRUE;
   FP_EN.Alarm_Low := TRUE;
   PWR := TRUE;
   EN_L := TRUE;
   OK := TRUE;
   AL_L := TRUE;
   AL_H := TRUE;
   WARN_L := TRUE;
   WARN_H := TRUE;
   MSW.EXT.Operation := TRUE;
   MSW.Status := 2;
   MSW.TimeStamp := 16#7EC8;
   BlockInfo.Ace_Version := 80;
   BlockInfo.Ace_BuildNo := 4;
   BlockInfo.State_Act := 2;
   BlockInfo.State_Prev := 202;
   BlockInfo.DB_Number := 2010;
   FP_PARM.EnableTime_Low_Acc := 5;
   FP_SIM.SIG_Enable := TRUE;
   FP_SIM.PWR_Enable := TRUE;
   ONS.SecPulse2 := TRUE;
   ONS.AL_L_Aux := TRUE;
   ONS.AL_H_Aux := TRUE;
   EnableTime_Low_Done := TRUE;
   StatusWork := 2;
   OUT.OK := TRUE;
   OUT.AL_L := TRUE;
   OUT.AL_H := TRUE;
   OUT.WARN_L := TRUE;
   OUT.WARN_H := TRUE;
   MSW_Status_Trans := 2;
END_DATA_BLOCK

DATA_BLOCK "_2010LV100F31E41_DB"   // DB2011
TITLE = Instance DB Alarm:
{ S7_Optimized_Access := 'FALSE' }
AUTHOR : METIS
NAME : ALARM_DB
VERSION : 8.0
// stored: InstanceOfName ACESYS_ALARM
"ACESYS_ALARM"
BEGIN
   FP_PARM.EnableTime_Low_Pre := 5;
   FP_EN.ParentSupress := TRUE;
   FP_EN.ParentSupressUnit := TRUE;
   FP_EN.Alarm_Low := TRUE;
   PWR := TRUE;
   EN_L := TRUE;
   OK := TRUE;
   AL_L := TRUE;
   AL_H := TRUE;
   WARN_L := TRUE;
   WARN_H := TRUE;
   MSW.EXT.Operation := TRUE;
   MSW.Status := 2;
   MSW.TimeStamp := 16#44F3;
   BlockInfo.Ace_Version := 80;
   BlockInfo.Ace_BuildNo := 4;
   BlockInfo.State_Act := 2;
   BlockInfo.State_Prev := 202;
   BlockInfo.DB_Number := 2011;
   FP_PARM.EnableTime_Low_Acc := 5;
   FP_SIM.SIG_Enable := TRUE;
   FP_SIM.PWR_Enable := TRUE;
   ONS.SecPulse2 := TRUE;
   ONS.AL_L_Aux := TRUE;
   ONS.AL_H_Aux := TRUE;
   EnableTime_Low_Done := TRUE;
   StatusWork := 2;
   OUT.OK := TRUE;
   OUT.AL_L := TRUE;
   OUT.AL_H := TRUE;
   OUT.WARN_L := TRUE;
   OUT.WARN_H := TRUE;
   MSW_Status_Trans := 2;
END_DATA_BLOCK

DATA_BLOCK "_2010LV100F41E41_DB"   // DB2012
TITLE = Instance DB Alarm:
{ S7_Optimized_Access := 'FALSE' }
AUTHOR : METIS
NAME : ALARM_DB
VERSION : 8.0
// stored: InstanceOfName ACESYS_ALARM
"ACESYS_ALARM"
BEGIN
   FP_PARM.EnableTime_Low_Pre := 5;
   FP_EN.ParentSupress := TRUE;
   FP_EN.ParentSupressUnit := TRUE;
   FP_EN.Alarm_Low := TRUE;
   PWR := TRUE;
   EN_L := TRUE;
   OK := TRUE;
   AL_L := TRUE;
   AL_H := TRUE;
   WARN_L := TRUE;
   WARN_H := TRUE;
   MSW.EXT.Operation := TRUE;
   MSW.Status := 2;
   MSW.TimeStamp := 16#7EC8;
   BlockInfo.Ace_Version := 80;
   BlockInfo.Ace_BuildNo := 4;
   BlockInfo.State_Act := 2;
   BlockInfo.State_Prev := 202;
   BlockInfo.DB_Number := 2012;
   FP_PARM.EnableTime_Low_Acc := 5;
   FP_SIM.SIG_Enable := TRUE;
   FP_SIM.PWR_Enable := TRUE;
   ONS.SecPulse2 := TRUE;
   ONS.AL_L_Aux := TRUE;
   ONS.AL_H_Aux := TRUE;
   EnableTime_Low_Done := TRUE;
   StatusWork := 2;
   OUT.OK := TRUE;
   OUT.AL_L := TRUE;
   OUT.AL_H := TRUE;
   OUT.WARN_L := TRUE;
   OUT.WARN_H := TRUE;
   MSW_Status_Trans := 2;
END_DATA_BLOCK

DATA_BLOCK "_2010CV300D02S41_DB"   // DB2013
TITLE = Instance DB Alarm:
{ S7_Optimized_Access := 'FALSE' }
AUTHOR : METIS
NAME : ALARM_DB
VERSION : 8.0
// stored: InstanceOfName ACESYS_ALARM
"ACESYS_ALARM"
BEGIN
   FP_PARM.EnableTime_Low_Pre := 5;
   FP_EN.ParentSupress := TRUE;
   FP_EN.ParentSupressUnit := TRUE;
   FP_EN.Alarm_Low := TRUE;
   PWR := TRUE;
   EN_L := TRUE;
   OK := TRUE;
   AL_L := TRUE;
   AL_H := TRUE;
   WARN_L := TRUE;
   WARN_H := TRUE;
   MSW.EXT.Operation := TRUE;
   MSW.Status := 2;
   MSW.TimeStamp := 16#31AB;
   BlockInfo.Ace_Version := 80;
   BlockInfo.Ace_BuildNo := 4;
   BlockInfo.State_Act := 2;
   BlockInfo.State_Prev := 1;
   BlockInfo.DB_Number := 2013;
   FP_PARM.EnableTime_Low_Acc := 5;
   FP_SIM.SIG_Enable := TRUE;
   FP_SIM.PWR_Enable := TRUE;
   ONS.SecPulse2 := TRUE;
   ONS.AL_L_Aux := TRUE;
   ONS.AL_H_Aux := TRUE;
   EnableTime_Low_Done := TRUE;
   StatusWork := 2;
   OUT.OK := TRUE;
   OUT.AL_L := TRUE;
   OUT.AL_H := TRUE;
   OUT.WARN_L := TRUE;
   OUT.WARN_H := TRUE;
   MSW_Status_Trans := 2;
END_DATA_BLOCK

DATA_BLOCK "_2010UP100G01U41_DB"   // DB2014
{ S7_Optimized_Access := 'FALSE' }
AUTHOR : FLSmidth
FAMILY : ACESYS
NAME : ALARM
VERSION : 8.0
// stored: InstanceOfName ACESYS_ALARM
"ACESYS_ALARM"
BEGIN
   PWR := TRUE;
   EN_L := TRUE;
   OK := TRUE;
   AL_L := TRUE;
   AL_H := TRUE;
   WARN_L := TRUE;
   WARN_H := TRUE;
   MSW.EXT.Operation := TRUE;
   MSW.Status := 2;
   MSW.TimeStamp := 16#32E8;
   BlockInfo.Ace_Version := 80;
   BlockInfo.Ace_BuildNo := 4;
   BlockInfo.State_Act := 2;
   BlockInfo.State_Prev := 202;
   BlockInfo.DB_Number := 2014;
   FP_EN.Alarm_Low := TRUE;
   FP_SIM.SIG_Enable := TRUE;
   FP_SIM.PWR_Enable := TRUE;
   ONS.SecPulse1 := TRUE;
   ONS.AL_L_Aux := TRUE;
   ONS.AL_H_Aux := TRUE;
   EnableTime_Low_Done := TRUE;
   Sec_Pulse := TRUE;
   StatusWork := 2;
   OUT.OK := TRUE;
   OUT.AL_L := TRUE;
   OUT.AL_H := TRUE;
   OUT.WARN_L := TRUE;
   OUT.WARN_H := TRUE;
   MSW_Status_Trans := 2;
END_DATA_BLOCK

DATA_BLOCK "_2010UP100G01U42_DB"   // DB2015
{ S7_Optimized_Access := 'FALSE' }
AUTHOR : FLSmidth
FAMILY : ACESYS
NAME : ALARM
VERSION : 8.0
// stored: InstanceOfName ACESYS_ALARM
"ACESYS_ALARM"
BEGIN
   PWR := TRUE;
   EN_L := TRUE;
   OK := TRUE;
   AL_L := TRUE;
   AL_H := TRUE;
   WARN_L := TRUE;
   WARN_H := TRUE;
   MSW.EXT.Operation := TRUE;
   MSW.Status := 2;
   MSW.TimeStamp := 16#32E8;
   BlockInfo.Ace_Version := 80;
   BlockInfo.Ace_BuildNo := 4;
   BlockInfo.State_Act := 2;
   BlockInfo.State_Prev := 202;
   BlockInfo.DB_Number := 2015;
   FP_EN.Alarm_Low := TRUE;
   FP_SIM.SIG_Enable := TRUE;
   FP_SIM.PWR_Enable := TRUE;
   ONS.SecPulse1 := TRUE;
   ONS.AL_L_Aux := TRUE;
   ONS.AL_H_Aux := TRUE;
   EnableTime_Low_Done := TRUE;
   Sec_Pulse := TRUE;
   StatusWork := 2;
   OUT.OK := TRUE;
   OUT.AL_L := TRUE;
   OUT.AL_H := TRUE;
   OUT.WARN_L := TRUE;
   OUT.WARN_H := TRUE;
   MSW_Status_Trans := 2;
END_DATA_BLOCK

DATA_BLOCK "_2010CV300D20Z42_DB"   // DB2016
{ S7_Optimized_Access := 'FALSE' }
AUTHOR : FLSmidth
FAMILY : ACESYS
NAME : ALARM
VERSION : 8.0
// stored: InstanceOfName ACESYS_ALARM
"ACESYS_ALARM"
BEGIN
   PWR := TRUE;
   EN_L := TRUE;
   OK := TRUE;
   AL_L := TRUE;
   AL_H := TRUE;
   WARN_L := TRUE;
   WARN_H := TRUE;
   MSW.EXT.Operation := TRUE;
   MSW.Status := 2;
   MSW.TimeStamp := 16#690C;
   BlockInfo.Ace_Version := 80;
   BlockInfo.Ace_BuildNo := 4;
   BlockInfo.State_Act := 2;
   BlockInfo.State_Prev := 202;
   BlockInfo.DB_Number := 2016;
   FP_EN.Alarm_Low := TRUE;
   FP_SIM.SIG_Enable := TRUE;
   FP_SIM.PWR_Enable := TRUE;
   ONS.SecPulse1 := TRUE;
   ONS.AL_L_Aux := TRUE;
   ONS.AL_H_Aux := TRUE;
   EnableTime_Low_Done := TRUE;
   Sec_Pulse := TRUE;
   StatusWork := 2;
   OUT.OK := TRUE;
   OUT.AL_L := TRUE;
   OUT.AL_H := TRUE;
   OUT.WARN_L := TRUE;
   OUT.WARN_H := TRUE;
   MSW_Status_Trans := 2;
END_DATA_BLOCK

DATA_BLOCK "_2010CV300D19Z42_DB"   // DB2017
{ S7_Optimized_Access := 'FALSE' }
AUTHOR : FLSmidth
FAMILY : ACESYS
NAME : ALARM
VERSION : 8.0
// stored: InstanceOfName ACESYS_ALARM
"ACESYS_ALARM"
BEGIN
   PWR := TRUE;
   EN_L := TRUE;
   OK := TRUE;
   AL_L := TRUE;
   AL_H := TRUE;
   WARN_L := TRUE;
   WARN_H := TRUE;
   MSW.EXT.Operation := TRUE;
   MSW.Status := 2;
   MSW.TimeStamp := 16#4583;
   BlockInfo.Ace_Version := 80;
   BlockInfo.Ace_BuildNo := 4;
   BlockInfo.State_Act := 2;
   BlockInfo.State_Prev := 202;
   BlockInfo.DB_Number := 2017;
   FP_EN.Alarm_Low := TRUE;
   FP_SIM.SIG_Enable := TRUE;
   FP_SIM.PWR_Enable := TRUE;
   ONS.SecPulse1 := TRUE;
   ONS.AL_L_Aux := TRUE;
   ONS.AL_H_Aux := TRUE;
   EnableTime_Low_Done := TRUE;
   StatusWork := 2;
   OUT.OK := TRUE;
   OUT.AL_L := TRUE;
   OUT.AL_H := TRUE;
   OUT.WARN_L := TRUE;
   OUT.WARN_H := TRUE;
   MSW_Status_Trans := 2;
END_DATA_BLOCK

DATA_BLOCK "_2010CV300D20Z41_DB"   // DB2018
{ S7_Optimized_Access := 'FALSE' }
AUTHOR : FLSmidth
FAMILY : ACESYS
NAME : ALARM
VERSION : 8.0
// stored: InstanceOfName ACESYS_ALARM
"ACESYS_ALARM"
BEGIN
   PWR := TRUE;
   EN_L := TRUE;
   OK := TRUE;
   AL_L := TRUE;
   AL_H := TRUE;
   WARN_L := TRUE;
   WARN_H := TRUE;
   MSW.EXT.Operation := TRUE;
   MSW.Status := 2;
   MSW.TimeStamp := 16#8915;
   BlockInfo.Ace_Version := 80;
   BlockInfo.Ace_BuildNo := 4;
   BlockInfo.State_Act := 2;
   BlockInfo.State_Prev := 202;
   BlockInfo.DB_Number := 2018;
   FP_EN.Alarm_Low := TRUE;
   FP_SIM.SIG_Enable := TRUE;
   FP_SIM.PWR_Enable := TRUE;
   ONS.SecPulse1 := TRUE;
   ONS.AL_L_Aux := TRUE;
   ONS.AL_H_Aux := TRUE;
   EnableTime_Low_Done := TRUE;
   StatusWork := 2;
   OUT.OK := TRUE;
   OUT.AL_L := TRUE;
   OUT.AL_H := TRUE;
   OUT.WARN_L := TRUE;
   OUT.WARN_H := TRUE;
   MSW_Status_Trans := 2;
END_DATA_BLOCK

DATA_BLOCK "_2010CV300D19Z41_DB"   // DB2019
{ S7_Optimized_Access := 'FALSE' }
AUTHOR : FLSmidth
FAMILY : ACESYS
NAME : ALARM
VERSION : 8.0
// stored: InstanceOfName ACESYS_ALARM
"ACESYS_ALARM"
BEGIN
   PWR := TRUE;
   EN_L := TRUE;
   OK := TRUE;
   AL_L := TRUE;
   AL_H := TRUE;
   WARN_L := TRUE;
   WARN_H := TRUE;
   MSW.EXT.Operation := TRUE;
   MSW.Status := 2;
   MSW.TimeStamp := 16#CF8D;
   BlockInfo.Ace_Version := 80;
   BlockInfo.Ace_BuildNo := 4;
   BlockInfo.State_Act := 2;
   BlockInfo.State_Prev := 1;
   BlockInfo.DB_Number := 2019;
   FP_EN.Alarm_Low := TRUE;
   FP_SIM.SIG_Enable := TRUE;
   FP_SIM.PWR_Enable := TRUE;
   ONS.SecPulse1 := TRUE;
   ONS.AL_L_Aux := TRUE;
   ONS.AL_H_Aux := TRUE;
   EnableTime_Low_Done := TRUE;
   StatusWork := 2;
   OUT.OK := TRUE;
   OUT.AL_L := TRUE;
   OUT.AL_H := TRUE;
   OUT.WARN_L := TRUE;
   OUT.WARN_H := TRUE;
   MSW_Status_Trans := 2;
END_DATA_BLOCK

DATA_BLOCK "_2010CV180OAC01_DB"   // DB2020
TITLE = Instance DB Alarm: _2010CV180OAC01
{ S7_Optimized_Access := 'FALSE' }
AUTHOR : METIS
NAME : ALARM_DB
VERSION : 8.0
// stored: InstanceOfName ACESYS_ALARM
"ACESYS_ALARM"
BEGIN
   FP_PARM.EnableTime_Low_Pre := 5;
   FP_EN.Alarm_Low := TRUE;
   PWR := TRUE;
   EN_L := TRUE;
   OK := TRUE;
   AL_L := TRUE;
   AL_H := TRUE;
   WARN_L := TRUE;
   WARN_H := TRUE;
   MSW.EXT.Operation := TRUE;
   MSW.Status := 2;
   MSW.TimeStamp := 16#B58B;
   BlockInfo.Ace_Version := 80;
   BlockInfo.Ace_BuildNo := 4;
   BlockInfo.State_Act := 2;
   BlockInfo.State_Prev := 202;
   BlockInfo.DB_Number := 2020;
   FP_PARM.EnableTime_Low_Acc := 5;
   FP_SIM.SIG_Enable := TRUE;
   FP_SIM.PWR_Enable := TRUE;
   ONS.SecPulse1 := TRUE;
   ONS.AL_L_Aux := TRUE;
   ONS.AL_H_Aux := TRUE;
   EnableTime_Low_Done := TRUE;
   StatusWork := 2;
   OUT.OK := TRUE;
   OUT.AL_L := TRUE;
   OUT.AL_H := TRUE;
   OUT.WARN_L := TRUE;
   OUT.WARN_H := TRUE;
   MSW_Status_Trans := 2;
END_DATA_BLOCK

DATA_BLOCK "_2010CV180YSQ01_DB"   // DB2021
TITLE = Instance DB Alarm: _2010CV180YSQ01_DB
{ S7_Optimized_Access := 'FALSE' }
AUTHOR : METIS
NAME : ALARM_DB
VERSION : 8.0
// stored: InstanceOfName ACESYS_ALARM
"ACESYS_ALARM"
BEGIN
   FP_PARM.EnableTime_Low_Pre := 5;
   FP_EN.ParentSupress := TRUE;
   FP_EN.ParentSupressUnit := TRUE;
   FP_EN.Alarm_Low := TRUE;
   PWR := TRUE;
   EN_L := TRUE;
   OK := TRUE;
   AL_L := TRUE;
   AL_H := TRUE;
   WARN_L := TRUE;
   WARN_H := TRUE;
   MSW.EXT.Operation := TRUE;
   MSW.Status := 2;
   MSW.TimeStamp := 16#7EC5;
   BlockInfo.Ace_Version := 80;
   BlockInfo.Ace_BuildNo := 4;
   BlockInfo.State_Act := 2;
   BlockInfo.State_Prev := 202;
   BlockInfo.DB_Number := 2021;
   FP_PARM.EnableTime_Low_Acc := 5;
   FP_SIM.SIG_Enable := TRUE;
   FP_SIM.PWR_Enable := TRUE;
   ONS.SecPulse1 := TRUE;
   ONS.AL_L_Aux := TRUE;
   ONS.AL_H_Aux := TRUE;
   EnableTime_Low_Done := TRUE;
   StatusWork := 2;
   OUT.OK := TRUE;
   OUT.AL_L := TRUE;
   OUT.AL_H := TRUE;
   OUT.WARN_L := TRUE;
   OUT.WARN_H := TRUE;
   MSW_Status_Trans := 2;
END_DATA_BLOCK

DATA_BLOCK "_2010CV180YAT01_DB"   // DB2022
TITLE = Instance DB Alarm: _2010CV180LSHH01_DB
{ S7_Optimized_Access := 'FALSE' }
AUTHOR : METIS
NAME : ALARM_DB
VERSION : 8.0
// stored: InstanceOfName ACESYS_ALARM
"ACESYS_ALARM"
BEGIN
   FP_PARM.EnableTime_Low_Pre := 5;
   FP_EN.Alarm_Low := TRUE;
   PWR := TRUE;
   EN_L := TRUE;
   OK := TRUE;
   AL_L := TRUE;
   AL_H := TRUE;
   WARN_L := TRUE;
   WARN_H := TRUE;
   MSW.EXT.Operation := TRUE;
   MSW.Status := 2;
   MSW.TimeStamp := 16#6A88;
   BlockInfo.Ace_Version := 80;
   BlockInfo.Ace_BuildNo := 4;
   BlockInfo.State_Act := 2;
   BlockInfo.State_Prev := 202;
   BlockInfo.DB_Number := 2022;
   FP_PARM.EnableTime_Low_Acc := 5;
   FP_SIM.SIG_Enable := TRUE;
   FP_SIM.PWR_Enable := TRUE;
   ONS.SecPulse1 := TRUE;
   ONS.AL_L_Aux := TRUE;
   ONS.AL_H_Aux := TRUE;
   EnableTime_Low_Done := TRUE;
   StatusWork := 2;
   OUT.OK := TRUE;
   OUT.AL_L := TRUE;
   OUT.AL_H := TRUE;
   OUT.WARN_L := TRUE;
   OUT.WARN_H := TRUE;
   MSW_Status_Trans := 2;
END_DATA_BLOCK

DATA_BLOCK "_2010CV180LSHH01_DB"   // DB2023
TITLE = Instance DB Alarm: _2010CV180LSHH01_DB
{ S7_Optimized_Access := 'FALSE' }
AUTHOR : METIS
NAME : ALARM_DB
VERSION : 8.0
// stored: InstanceOfName ACESYS_ALARM
"ACESYS_ALARM"
BEGIN
   FP_PARM.EnableTime_Low_Pre := 5;
   FP_EN.Alarm_Low := TRUE;
   PWR := TRUE;
   EN_L := TRUE;
   OK := TRUE;
   AL_L := TRUE;
   AL_H := TRUE;
   WARN_L := TRUE;
   WARN_H := TRUE;
   MSW.EXT.Operation := TRUE;
   MSW.Status := 2;
   MSW.TimeStamp := 16#25CC;
   BlockInfo.Ace_Version := 80;
   BlockInfo.Ace_BuildNo := 4;
   BlockInfo.State_Act := 2;
   BlockInfo.State_Prev := 202;
   BlockInfo.DB_Number := 2023;
   FP_PARM.EnableTime_Low_Acc := 5;
   FP_SIM.SIG_Enable := TRUE;
   FP_SIM.PWR_Enable := TRUE;
   ONS.SecPulse1 := TRUE;
   ONS.AL_L_Aux := TRUE;
   ONS.AL_H_Aux := TRUE;
   EnableTime_Low_Done := TRUE;
   StatusWork := 2;
   OUT.OK := TRUE;
   OUT.AL_L := TRUE;
   OUT.AL_H := TRUE;
   OUT.WARN_L := TRUE;
   OUT.WARN_H := TRUE;
   MSW_Status_Trans := 2;
END_DATA_BLOCK

DATA_BLOCK "_2010CV120OAC01_DB"   // DB2024
TITLE = Instance DB Alarm: _2010CV180OAC01
{ S7_Optimized_Access := 'FALSE' }
AUTHOR : METIS
NAME : ALARM_DB
VERSION : 8.0
// stored: InstanceOfName ACESYS_ALARM
"ACESYS_ALARM"
BEGIN
   FP_PARM.EnableTime_Low_Pre := 5;
   FP_EN.Alarm_Low := TRUE;
   PWR := TRUE;
   EN_L := TRUE;
   OK := TRUE;
   AL_L := TRUE;
   AL_H := TRUE;
   WARN_L := TRUE;
   WARN_H := TRUE;
   MSW.EXT.Operation := TRUE;
   MSW.Status := 2;
   MSW.TimeStamp := 16#6963;
   BlockInfo.Ace_Version := 80;
   BlockInfo.Ace_BuildNo := 4;
   BlockInfo.State_Act := 2;
   BlockInfo.State_Prev := 202;
   BlockInfo.DB_Number := 2024;
   FP_PARM.EnableTime_Low_Acc := 5;
   FP_SIM.SIG_Enable := TRUE;
   FP_SIM.PWR_Enable := TRUE;
   ONS.SecPulse1 := TRUE;
   ONS.AL_L_Aux := TRUE;
   ONS.AL_H_Aux := TRUE;
   EnableTime_Low_Done := TRUE;
   StatusWork := 2;
   OUT.OK := TRUE;
   OUT.AL_L := TRUE;
   OUT.AL_H := TRUE;
   OUT.WARN_L := TRUE;
   OUT.WARN_H := TRUE;
   MSW_Status_Trans := 2;
END_DATA_BLOCK

DATA_BLOCK "_2010CV120YSQ01_DB"   // DB2025
TITLE = Instance DB Alarm: _2010CV180YSQ01_DB
{ S7_Optimized_Access := 'FALSE' }
AUTHOR : 7Art
NAME : ALARM_DB
VERSION : 8.0
// stored: InstanceOfName ACESYS_ALARM
"ACESYS_ALARM"
BEGIN
   FP_PARM.EnableTime_Low_Pre := 5;
   FP_EN.ParentSupress := TRUE;
   FP_EN.ParentSupressUnit := TRUE;
   FP_EN.Alarm_Low := TRUE;
   PWR := TRUE;
   EN_L := TRUE;
   OK := TRUE;
   AL_L := TRUE;
   AL_H := TRUE;
   WARN_L := TRUE;
   WARN_H := TRUE;
   MSW.EXT.Operation := TRUE;
   MSW.Status := 2;
   MSW.TimeStamp := 16#90A2;
   BlockInfo.Ace_Version := 80;
   BlockInfo.Ace_BuildNo := 4;
   BlockInfo.State_Act := 2;
   BlockInfo.State_Prev := 202;
   BlockInfo.DB_Number := 2025;
   FP_PARM.EnableTime_Low_Acc := 5;
   FP_SIM.SIG_Enable := TRUE;
   FP_SIM.PWR_Enable := TRUE;
   ONS.SecPulse1 := TRUE;
   ONS.AL_L_Aux := TRUE;
   ONS.AL_H_Aux := TRUE;
   EnableTime_Low_Done := TRUE;
   StatusWork := 2;
   OUT.OK := TRUE;
   OUT.AL_L := TRUE;
   OUT.AL_H := TRUE;
   OUT.WARN_L := TRUE;
   OUT.WARN_H := TRUE;
   MSW_Status_Trans := 2;
END_DATA_BLOCK

DATA_BLOCK "_2010OB190YSES01_DB"   // DB2026
TITLE = Instance DB Alarm: _2010OB190YSES01_DB Safety relay
{ S7_Optimized_Access := 'FALSE' }
AUTHOR : 7Art
NAME : ALARM_DB
VERSION : 8.0
// stored: InstanceOfName ACESYS_ALARM
"ACESYS_ALARM"
BEGIN
   FP_PARM.EnableTime_Low_Pre := 5;
   FP_EN.ParentSupress := TRUE;
   FP_EN.ParentSupressUnit := TRUE;
   FP_EN.Alarm_Low := TRUE;
   PWR := TRUE;
   EN_L := TRUE;
   OK := TRUE;
   AL_L := TRUE;
   AL_H := TRUE;
   WARN_L := TRUE;
   WARN_H := TRUE;
   MSW.EXT.Operation := TRUE;
   MSW.Status := 2;
   MSW.TimeStamp := 16#61B4;
   BlockInfo.Ace_Version := 80;
   BlockInfo.Ace_BuildNo := 4;
   BlockInfo.State_Act := 2;
   BlockInfo.State_Prev := 202;
   BlockInfo.DB_Number := 2026;
   FP_PARM.EnableTime_Low_Acc := 5;
   FP_SIM.SIG_Enable := TRUE;
   FP_SIM.PWR_Enable := TRUE;
   ONS.SecPulse1 := TRUE;
   ONS.AL_L_Aux := TRUE;
   ONS.AL_H_Aux := TRUE;
   EnableTime_Low_Done := TRUE;
   StatusWork := 2;
   OUT.OK := TRUE;
   OUT.AL_L := TRUE;
   OUT.AL_H := TRUE;
   OUT.WARN_L := TRUE;
   OUT.WARN_H := TRUE;
   MSW_Status_Trans := 2;
END_DATA_BLOCK

DATA_BLOCK "_2010OB190OAC01_DB"   // DB2027
TITLE = Instance DB Alarm: _2010OB190OAC01_DB Emergency stop
{ S7_Optimized_Access := 'FALSE' }
AUTHOR : 7Art
NAME : ALARM_DB
VERSION : 8.0
// stored: InstanceOfName ACESYS_ALARM
"ACESYS_ALARM"
BEGIN
   FP_PARM.EnableTime_Low_Pre := 5;
   FP_EN.ParentSupress := TRUE;
   FP_EN.ParentSupressUnit := TRUE;
   FP_EN.Alarm_Low := TRUE;
   PWR := TRUE;
   EN_L := TRUE;
   OK := TRUE;
   AL_L := TRUE;
   AL_H := TRUE;
   WARN_L := TRUE;
   WARN_H := TRUE;
   MSW.EXT.Operation := TRUE;
   MSW.Status := 2;
   MSW.TimeStamp := 16#72EA;
   BlockInfo.Ace_Version := 80;
   BlockInfo.Ace_BuildNo := 4;
   BlockInfo.State_Act := 2;
   BlockInfo.State_Prev := 202;
   BlockInfo.DB_Number := 2027;
   FP_PARM.EnableTime_Low_Acc := 5;
   FP_SIM.SIG_Enable := TRUE;
   FP_SIM.PWR_Enable := TRUE;
   ONS.SecPulse1 := TRUE;
   ONS.AL_L_Aux := TRUE;
   ONS.AL_H_Aux := TRUE;
   EnableTime_Low_Done := TRUE;
   StatusWork := 2;
   OUT.OK := TRUE;
   OUT.AL_L := TRUE;
   OUT.AL_H := TRUE;
   OUT.WARN_L := TRUE;
   OUT.WARN_H := TRUE;
   MSW_Status_Trans := 2;
END_DATA_BLOCK

DATA_BLOCK "_2010OB190YSQ01_DB"   // DB2028
TITLE = Instance DB Alarm: 2010OB190YSQ01 Breaker feedback
{ S7_Optimized_Access := 'FALSE' }
AUTHOR : 7Art
NAME : ALARM_DB
VERSION : 8.0
// stored: InstanceOfName ACESYS_ALARM
"ACESYS_ALARM"
BEGIN
   FP_PARM.EnableTime_Low_Pre := 5;
   FP_EN.ParentSupress := TRUE;
   FP_EN.ParentSupressUnit := TRUE;
   FP_EN.Alarm_Low := TRUE;
   PWR := TRUE;
   EN_L := TRUE;
   OK := TRUE;
   AL_L := TRUE;
   AL_H := TRUE;
   WARN_L := TRUE;
   WARN_H := TRUE;
   MSW.EXT.Operation := TRUE;
   MSW.Status := 2;
   MSW.TimeStamp := 16#906C;
   BlockInfo.Ace_Version := 80;
   BlockInfo.Ace_BuildNo := 4;
   BlockInfo.State_Act := 2;
   BlockInfo.State_Prev := 202;
   BlockInfo.DB_Number := 2028;
   FP_PARM.EnableTime_Low_Acc := 5;
   FP_SIM.SIG_Enable := TRUE;
   FP_SIM.PWR_Enable := TRUE;
   ONS.SecPulse1 := TRUE;
   ONS.AL_L_Aux := TRUE;
   ONS.AL_H_Aux := TRUE;
   EnableTime_Low_Done := TRUE;
   StatusWork := 2;
   OUT.OK := TRUE;
   OUT.AL_L := TRUE;
   OUT.AL_H := TRUE;
   OUT.WARN_L := TRUE;
   OUT.WARN_H := TRUE;
   MSW_Status_Trans := 2;
END_DATA_BLOCK

DATA_BLOCK "_2010OB190YSK01_DB"   // DB2029
TITLE = Instance DB Alarm: 2010OB190YSK01 Contractor feedback
{ S7_Optimized_Access := 'FALSE' }
AUTHOR : 7Art
NAME : ALARM_DB
VERSION : 8.0
// stored: InstanceOfName ACESYS_ALARM
"ACESYS_ALARM"
BEGIN
   FP_PARM.EnableTime_Low_Pre := 5;
   FP_EN.ParentSupress := TRUE;
   FP_EN.ParentSupressUnit := TRUE;
   FP_EN.Alarm_Low := TRUE;
   PWR := TRUE;
   EN_L := TRUE;
   OK := TRUE;
   AL_L := TRUE;
   AL_H := TRUE;
   WARN_L := TRUE;
   WARN_H := TRUE;
   MSW.EXT.Operation := TRUE;
   MSW.Status := 2;
   MSW.TimeStamp := 16#906C;
   BlockInfo.Ace_Version := 80;
   BlockInfo.Ace_BuildNo := 4;
   BlockInfo.State_Act := 2;
   BlockInfo.State_Prev := 202;
   BlockInfo.DB_Number := 2029;
   FP_PARM.EnableTime_Low_Acc := 5;
   FP_SIM.SIG_Enable := TRUE;
   FP_SIM.PWR_Enable := TRUE;
   ONS.SecPulse1 := TRUE;
   ONS.AL_L_Aux := TRUE;
   ONS.AL_H_Aux := TRUE;
   EnableTime_Low_Done := TRUE;
   StatusWork := 2;
   OUT.OK := TRUE;
   OUT.AL_L := TRUE;
   OUT.AL_H := TRUE;
   OUT.WARN_L := TRUE;
   OUT.WARN_H := TRUE;
   MSW_Status_Trans := 2;
END_DATA_BLOCK

DATA_BLOCK "_2010OB190SW01_DB"   // DB2030
TITLE = Instance DB Alarm: 2010OB190SW01 Isolator switch
{ S7_Optimized_Access := 'FALSE' }
AUTHOR : 7Art
NAME : ALARM_DB
VERSION : 8.0
// stored: InstanceOfName ACESYS_ALARM
"ACESYS_ALARM"
BEGIN
   FP_PARM.EnableTime_Low_Pre := 5;
   FP_EN.ParentSupress := TRUE;
   FP_EN.ParentSupressUnit := TRUE;
   FP_EN.Alarm_Low := TRUE;
   PWR := TRUE;
   EN_L := TRUE;
   OK := TRUE;
   AL_L := TRUE;
   AL_H := TRUE;
   WARN_L := TRUE;
   WARN_H := TRUE;
   MSW.EXT.Operation := TRUE;
   MSW.Status := 2;
   MSW.TimeStamp := 16#72EA;
   BlockInfo.Ace_Version := 80;
   BlockInfo.Ace_BuildNo := 4;
   BlockInfo.State_Act := 2;
   BlockInfo.State_Prev := 202;
   BlockInfo.DB_Number := 2030;
   FP_PARM.EnableTime_Low_Acc := 5;
   FP_SIM.SIG_Enable := TRUE;
   FP_SIM.PWR_Enable := TRUE;
   ONS.SecPulse1 := TRUE;
   ONS.AL_L_Aux := TRUE;
   ONS.AL_H_Aux := TRUE;
   EnableTime_Low_Done := TRUE;
   StatusWork := 2;
   OUT.OK := TRUE;
   OUT.AL_L := TRUE;
   OUT.AL_H := TRUE;
   OUT.WARN_L := TRUE;
   OUT.WARN_H := TRUE;
   MSW_Status_Trans := 2;
END_DATA_BLOCK

DATA_BLOCK "_2010OB190USF01_DB"   // DB2031
TITLE = Instance DB Alarm: 2010OB190USF01 Healthy Box
{ S7_Optimized_Access := 'FALSE' }
AUTHOR : 7Art
NAME : ALARM_DB
VERSION : 8.0
// stored: InstanceOfName ACESYS_ALARM
"ACESYS_ALARM"
BEGIN
   FP_PARM.EnableTime_Low_Pre := 5;
   FP_EN.ParentSupress := TRUE;
   FP_EN.ParentSupressUnit := TRUE;
   FP_EN.Alarm_Low := TRUE;
   PWR := TRUE;
   EN_L := TRUE;
   OK := TRUE;
   AL_L := TRUE;
   AL_H := TRUE;
   WARN_L := TRUE;
   WARN_H := TRUE;
   MSW.EXT.Operation := TRUE;
   MSW.Status := 2;
   MSW.TimeStamp := 16#9071;
   BlockInfo.Ace_Version := 80;
   BlockInfo.Ace_BuildNo := 4;
   BlockInfo.State_Act := 2;
   BlockInfo.State_Prev := 202;
   BlockInfo.DB_Number := 2031;
   FP_PARM.EnableTime_Low_Acc := 5;
   FP_SIM.SIG_Enable := TRUE;
   FP_SIM.PWR_Enable := TRUE;
   ONS.SecPulse1 := TRUE;
   ONS.AL_L_Aux := TRUE;
   ONS.AL_H_Aux := TRUE;
   EnableTime_Low_Done := TRUE;
   StatusWork := 2;
   OUT.OK := TRUE;
   OUT.AL_L := TRUE;
   OUT.AL_H := TRUE;
   OUT.WARN_L := TRUE;
   OUT.WARN_H := TRUE;
   MSW_Status_Trans := 2;
END_DATA_BLOCK

DATA_BLOCK "_2010BF110U01OAC01_DB"   // DB2032
TITLE = Instance DB Alarm: 2010BF110U01OAC01 Emergency stop PB
{ S7_Optimized_Access := 'FALSE' }
AUTHOR : 7Art
NAME : ALARM_DB
VERSION : 8.0
// stored: InstanceOfName ACESYS_ALARM
"ACESYS_ALARM"
BEGIN
   FP_PARM.EnableTime_Low_Pre := 5;
   FP_EN.Alarm_Low := TRUE;
   PWR := TRUE;
   EN_L := TRUE;
   OK := TRUE;
   AL_L := TRUE;
   AL_H := TRUE;
   WARN_L := TRUE;
   WARN_H := TRUE;
   MSW.EXT.Operation := TRUE;
   MSW.Status := 2;
   MSW.TimeStamp := 16#9376;
   BlockInfo.Ace_Version := 80;
   BlockInfo.Ace_BuildNo := 4;
   BlockInfo.State_Act := 2;
   BlockInfo.State_Prev := 202;
   BlockInfo.DB_Number := 2032;
   FP_PARM.EnableTime_Low_Acc := 5;
   FP_SIM.SIG_Enable := TRUE;
   FP_SIM.PWR_Enable := TRUE;
   ONS.SecPulse1 := TRUE;
   ONS.AL_L_Aux := TRUE;
   ONS.AL_H_Aux := TRUE;
   EnableTime_Low_Done := TRUE;
   StatusWork := 2;
   OUT.OK := TRUE;
   OUT.AL_L := TRUE;
   OUT.AL_H := TRUE;
   OUT.WARN_L := TRUE;
   OUT.WARN_H := TRUE;
   MSW_Status_Trans := 2;
END_DATA_BLOCK

DATA_BLOCK "_2010BF110U01OAC02_DB"   // DB2033
TITLE = Instance DB Alarm: 2010BF110U01OAC02 Emergency stop PB
{ S7_Optimized_Access := 'FALSE' }
AUTHOR : 7Art
NAME : ALARM_DB
VERSION : 8.0
// stored: InstanceOfName ACESYS_ALARM
"ACESYS_ALARM"
BEGIN
   FP_PARM.EnableTime_Low_Pre := 5;
   FP_EN.Alarm_Low := TRUE;
   PWR := TRUE;
   EN_L := TRUE;
   OK := TRUE;
   AL_L := TRUE;
   AL_H := TRUE;
   WARN_L := TRUE;
   WARN_H := TRUE;
   MSW.EXT.Operation := TRUE;
   MSW.Status := 2;
   MSW.TimeStamp := 16#6BF5;
   BlockInfo.Ace_Version := 80;
   BlockInfo.Ace_BuildNo := 4;
   BlockInfo.State_Act := 2;
   BlockInfo.State_Prev := 1;
   BlockInfo.DB_Number := 2033;
   FP_PARM.EnableTime_Low_Acc := 5;
   FP_SIM.SIG_Enable := TRUE;
   FP_SIM.PWR_Enable := TRUE;
   ONS.SecPulse1 := TRUE;
   ONS.AL_L_Aux := TRUE;
   ONS.AL_H_Aux := TRUE;
   EnableTime_Low_Done := TRUE;
   StatusWork := 2;
   OUT.OK := TRUE;
   OUT.AL_L := TRUE;
   OUT.AL_H := TRUE;
   OUT.WARN_L := TRUE;
   OUT.WARN_H := TRUE;
   MSW_Status_Trans := 2;
END_DATA_BLOCK

DATA_BLOCK "_2010BF110U01OAC03_DB"   // DB2034
TITLE = Instance DB Alarm: 2010BF110U01OAC03 Emergency stop PB
{ S7_Optimized_Access := 'FALSE' }
AUTHOR : 7Art
NAME : ALARM_DB
VERSION : 8.0
// stored: InstanceOfName ACESYS_ALARM
"ACESYS_ALARM"
BEGIN
   FP_PARM.EnableTime_Low_Pre := 5;
   FP_EN.Alarm_Low := TRUE;
   PWR := TRUE;
   EN_L := TRUE;
   OK := TRUE;
   AL_L := TRUE;
   AL_H := TRUE;
   WARN_L := TRUE;
   WARN_H := TRUE;
   MSW.EXT.Operation := TRUE;
   MSW.Status := 2;
   MSW.TimeStamp := 16#2F28;
   BlockInfo.Ace_Version := 80;
   BlockInfo.Ace_BuildNo := 4;
   BlockInfo.State_Act := 2;
   BlockInfo.State_Prev := 202;
   BlockInfo.DB_Number := 2034;
   FP_PARM.EnableTime_Low_Acc := 5;
   FP_SIM.SIG_Enable := TRUE;
   FP_SIM.PWR_Enable := TRUE;
   ONS.SecPulse1 := TRUE;
   ONS.AL_L_Aux := TRUE;
   ONS.AL_H_Aux := TRUE;
   EnableTime_Low_Done := TRUE;
   StatusWork := 2;
   OUT.OK := TRUE;
   OUT.AL_L := TRUE;
   OUT.AL_H := TRUE;
   OUT.WARN_L := TRUE;
   OUT.WARN_H := TRUE;
   MSW_Status_Trans := 2;
END_DATA_BLOCK

DATA_BLOCK "_2010BF110U01YSQ01_DB"   // DB2035
TITLE = Instance DB Alarm: 2010BF110U01YSQ01 Breaker feedback
{ S7_Optimized_Access := 'FALSE' }
AUTHOR : 7Art
NAME : ALARM_DB
VERSION : 8.0
// stored: InstanceOfName ACESYS_ALARM
"ACESYS_ALARM"
BEGIN
   FP_PARM.EnableTime_Low_Pre := 5;
   FP_EN.Alarm_Low := TRUE;
   PWR := TRUE;
   EN_L := TRUE;
   OK := TRUE;
   AL_L := TRUE;
   AL_H := TRUE;
   WARN_L := TRUE;
   WARN_H := TRUE;
   MSW.EXT.Operation := TRUE;
   MSW.Status := 2;
   MSW.TimeStamp := 16#8E89;
   BlockInfo.Ace_Version := 80;
   BlockInfo.Ace_BuildNo := 4;
   BlockInfo.State_Act := 2;
   BlockInfo.State_Prev := 202;
   BlockInfo.DB_Number := 2035;
   FP_PARM.EnableTime_Low_Acc := 5;
   FP_SIM.SIG_Enable := TRUE;
   FP_SIM.PWR_Enable := TRUE;
   ONS.SecPulse1 := TRUE;
   ONS.AL_L_Aux := TRUE;
   ONS.AL_H_Aux := TRUE;
   EnableTime_Low_Done := TRUE;
   StatusWork := 2;
   OUT.OK := TRUE;
   OUT.AL_L := TRUE;
   OUT.AL_H := TRUE;
   OUT.WARN_L := TRUE;
   OUT.WARN_H := TRUE;
   MSW_Status_Trans := 2;
END_DATA_BLOCK

DATA_BLOCK "_2010SC130U01OAC01_DB"   // DB2036
TITLE = Instance DB Alarm: Emergency stop PB
{ S7_Optimized_Access := 'FALSE' }
AUTHOR : 7Art
NAME : ALARM_DB
VERSION : 8.0
// stored: InstanceOfName ACESYS_ALARM
"ACESYS_ALARM"
BEGIN
   FP_PARM.EnableTime_Low_Pre := 5;
   FP_EN.Alarm_Low := TRUE;
   PWR := TRUE;
   EN_L := TRUE;
   OK := TRUE;
   AL_L := TRUE;
   AL_H := TRUE;
   WARN_L := TRUE;
   WARN_H := TRUE;
   MSW.EXT.Operation := TRUE;
   MSW.Status := 2;
   MSW.TimeStamp := 16#A748;
   BlockInfo.Ace_Version := 80;
   BlockInfo.Ace_BuildNo := 4;
   BlockInfo.State_Act := 2;
   BlockInfo.State_Prev := 202;
   BlockInfo.DB_Number := 2036;
   FP_PARM.EnableTime_Low_Acc := 5;
   FP_SIM.SIG_Enable := TRUE;
   FP_SIM.PWR_Enable := TRUE;
   ONS.SecPulse1 := TRUE;
   ONS.AL_L_Aux := TRUE;
   ONS.AL_H_Aux := TRUE;
   EnableTime_Low_Done := TRUE;
   StatusWork := 2;
   OUT.OK := TRUE;
   OUT.AL_L := TRUE;
   OUT.AL_H := TRUE;
   OUT.WARN_L := TRUE;
   OUT.WARN_H := TRUE;
   MSW_Status_Trans := 2;
END_DATA_BLOCK

DATA_BLOCK "_2010SC130U01YSQ01_DB"   // DB2037
TITLE = Instance DB Alarm: Breaker feedback
{ S7_Optimized_Access := 'FALSE' }
AUTHOR : 7Art
NAME : ALARM_DB
VERSION : 8.0
// stored: InstanceOfName ACESYS_ALARM
"ACESYS_ALARM"
BEGIN
   FP_PARM.EnableTime_Low_Pre := 5;
   FP_EN.Alarm_Low := TRUE;
   PWR := TRUE;
   EN_L := TRUE;
   OK := TRUE;
   AL_L := TRUE;
   AL_H := TRUE;
   WARN_L := TRUE;
   WARN_H := TRUE;
   MSW.EXT.Operation := TRUE;
   MSW.Status := 2;
   MSW.TimeStamp := 16#8DD6;
   BlockInfo.Ace_Version := 80;
   BlockInfo.Ace_BuildNo := 4;
   BlockInfo.State_Act := 2;
   BlockInfo.State_Prev := 202;
   BlockInfo.DB_Number := 2037;
   FP_PARM.EnableTime_Low_Acc := 5;
   FP_SIM.SIG_Enable := TRUE;
   FP_SIM.PWR_Enable := TRUE;
   ONS.SecPulse1 := TRUE;
   ONS.AL_L_Aux := TRUE;
   ONS.AL_H_Aux := TRUE;
   EnableTime_Low_Done := TRUE;
   StatusWork := 2;
   OUT.OK := TRUE;
   OUT.AL_L := TRUE;
   OUT.AL_H := TRUE;
   OUT.WARN_L := TRUE;
   OUT.WARN_H := TRUE;
   MSW_Status_Trans := 2;
END_DATA_BLOCK

